gfCNCPoint4[12082] = {X 126.3568, Y 92.7333, Z -5.5000, A 0.000, B 0.000, C 0.000 }
gfCNCPoint4[12083] = {X 127.2181, Y 92.5238, Z -5.5000, A 0.000, B 0.000, C 0.000 }
gfCNCPoint4[12084] = {X 128.4710, Y 91.3461, Z -5.5000, A 0.000, B 0.000, C 0.000 }
gfCNCPoint4[12085] = {X 129.6569, Y 90.1009, Z -5.5000, A 0.000, B 0.000, C 0.000 }
gfCNCPoint4[12086] = {X 140.8575, Y 77.8010, Z -5.5000, A 0.000, B 0.000, C 0.000 }
gfCNCPoint4[12087] = {X 137.8975, Y 75.1055, Z -5.5000, A 0.000, B 0.000, C 0.000 }
gfCNCPoint4[12088] = {X 137.8979, Y 75.1051, Z -5.5000, A 0.000, B 0.000, C 0.000 }
gfCNCPoint4[12089] = {X 140.9141, Y 77.8526, Z -5.5000, A 0.000, B 0.000, C 0.000 }
gfCNCPoint4[12090] = {X 156.0371, Y 61.2507, Z -5.5000, A 0.000, B 0.000, C 0.000 }
gfCNCPoint4[12091] = {X 155.6323, Y 60.5351, Z -5.5000, A 0.000, B 0.000, C 0.000 }
gfCNCPoint4[12092] = {X 155.3824, Y 59.7518, Z -5.5000, A 0.000, B 0.000, C 0.000 }
gfCNCPoint4[12093] = {X 155.2980, Y 58.9341, Z -5.5000, A 0.000, B 0.000, C 0.000 }
gfCNCPoint4[12094] = {X 155.2980, Y 58.0000, Z -5.5000, A 0.000, B 0.000, C 0.000 }
gfCNCPoint4[12095] = {X 155.3982, Y 57.1099, Z -5.5000, A 0.000, B 0.000, C 0.000 }
gfCNCPoint4[12096] = {X 155.6941, Y 56.2645, Z -5.5000, A 0.000, B 0.000, C 0.000 }
gfCNCPoint4[12097] = {X 156.1706, Y 55.5060, Z -5.5000, A 0.000, B 0.000, C 0.000 }
gfCNCPoint4[12098] = {X 156.8040, Y 54.8727, Z -5.5000, A 0.000, B 0.000, C 0.000 }
gfCNCPoint4[12099] = {X 157.5624, Y 54.3961, Z -5.5000, A 0.000, B 0.000, C 0.000 }
gfCNCPoint4[12100] = {X 158.4079, Y 54.1003, Z -5.5000, A 0.000, B 0.000, C 0.000 }
gfCNCPoint4[12101] = {X 159.2980, Y 54.0000, Z -5.5000, A 0.000, B 0.000, C 0.000 }
gfCNCPoint4[12102] = {X 178.5335, Y 54.0000, Z -5.5000, A 0.000, B 0.000, C 0.000 }
gfCNCPoint4[12103] = {X 179.4236, Y 54.1003, Z -5.5000, A 0.000, B 0.000, C 0.000 }
gfCNCPoint4[12104] = {X 180.2690, Y 54.3961, Z -5.5000, A 0.000, B 0.000, C 0.000 }
gfCNCPoint4[12105] = {X 181.0275, Y 54.8727, Z -5.5000, A 0.000, B 0.000, C 0.000 }
gfCNCPoint4[12106] = {X 181.6608, Y 55.5060, Z -5.5000, A 0.000, B 0.000, C 0.000 }
gfCNCPoint4[12107] = {X 182.1374, Y 56.2645, Z -5.5000, A 0.000, B 0.000, C 0.000 }
gfCNCPoint4[12108] = {X 182.4332, Y 57.1099, Z -5.5000, A 0.000, B 0.000, C 0.000 }
gfCNCPoint4[12109] = {X 182.5335, Y 58.0000, Z -5.5000, A 0.000, B 0.000, C 0.000 }
gfCNCPoint4[12110] = {X 182.5334, Y 58.9671, Z -5.5000, A 0.000, B 0.000, C 0.000 }
gfCNCPoint4[12111] = {X 182.4463, Y 59.7646, Z -5.5000, A 0.000, B 0.000, C 0.000 }
gfCNCPoint4[12112] = {X 182.2019, Y 60.5286, Z -5.5000, A 0.000, B 0.000, C 0.000 }
gfCNCPoint4[12113] = {X 181.8100, Y 61.2285, Z -5.5000, A 0.000, B 0.000, C 0.000 }
gfCNCPoint4[12114] = {X 209.2433, Y 91.1704, Z -5.5000, A 0.000, B 0.000, C 0.000 }
gfCNCPoint4[12115] = {X 209.9164, Y 91.8534, Z -5.5000, A 0.000, B 0.000, C 0.000 }
gfCNCPoint4[12116] = {X 210.6375, Y 92.4856, Z -5.5000, A 0.000, B 0.000, C 0.000 }
gfCNCPoint4[12117] = {X 210.9790, Y 92.7012, Z -5.5000, A 0.000, B 0.000, C 0.000 }
gfCNCPoint4[12118] = {X 211.3621, Y 92.8295, Z -5.5000, A 0.000, B 0.000, C 0.000 }
gfCNCPoint4[12119] = {X 212.0545, Y 92.9775, Z -5.5000, A 0.000, B 0.000, C 0.000 }
gfCNCPoint4[12120] = {X 213.3961, Y 93.1465, Z -5.5000, A 0.000, B 0.000, C 0.000 }
gfCNCPoint4[12121] = {X 214.4555, Y 93.0562, Z -5.5000, A 0.000, B 0.000, C 0.000 }
gfCNCPoint4[12122] = {X 215.5170, Y 92.9951, Z -5.5000, A 0.000, B 0.000, C 0.000 }
gfCNCPoint4[12123] = {X 216.2444, Y 92.9150, Z -5.5000, A 0.000, B 0.000, C 0.000 }
gfCNCPoint4[12124] = {X 216.9448, Y 92.7028, Z -5.5000, A 0.000, B 0.000, C 0.000 }
gfCNCPoint4[12125] = {X 217.5944, Y 92.3657, Z -5.5000, A 0.000, B 0.000, C 0.000 }
gfCNCPoint4[12126] = {X 223.1343, Y 88.7905, Z -5.5000, A 0.000, B 0.000, C 0.000 }
gfCNCPoint4[12127] = {X 246.5290, Y 73.8310, Z -5.5000, A 0.000, B 0.000, C 0.000 }
gfCNCPoint4[12128] = {X 221.7493, Y 64.1069, Z -5.5000, A 0.000, B 0.000, C 0.000 }
gfCNCPoint4[12129] = {X 219.9471, Y 63.5037, Z -5.5000, A 0.000, B 0.000, C 0.000 }
gfCNCPoint4[12130] = {X 218.0879, Y 63.1103, Z -5.5000, A 0.000, B 0.000, C 0.000 }
gfCNCPoint4[12131] = {X 216.1958, Y 62.9318, Z -5.5000, A 0.000, B 0.000, C 0.000 }
gfCNCPoint4[12132] = {X 215.3283, Y 62.8064, Z -5.5000, A 0.000, B 0.000, C 0.000 }
gfCNCPoint4[12133] = {X 214.5089, Y 62.4951, Z -5.5000, A 0.000, B 0.000, C 0.000 }
gfCNCPoint4[12134] = {X 213.7770, Y 62.0127, Z -5.5000, A 0.000, B 0.000, C 0.000 }
gfCNCPoint4[12135] = {X 213.1677, Y 61.3825, Z -5.5000, A 0.000, B 0.000, C 0.000 }
gfCNCPoint4[12136] = {X 212.7104, Y 60.6348, Z -5.5000, A 0.000, B 0.000, C 0.000 }
gfCNCPoint4[12137] = {X 212.4268, Y 59.8053, Z -5.5000, A 0.000, B 0.000, C 0.000 }
gfCNCPoint4[12138] = {X 212.3308, Y 58.9341, Z -5.5000, A 0.000, B 0.000, C 0.000 }
gfCNCPoint4[12139] = {X 212.3308, Y 58.0000, Z -5.5000, A 0.000, B 0.000, C 0.000 }
gfCNCPoint4[12140] = {X 212.4311, Y 57.1099, Z -5.5000, A 0.000, B 0.000, C 0.000 }
gfCNCPoint4[12141] = {X 212.7269, Y 56.2645, Z -5.5000, A 0.000, B 0.000, C 0.000 }
gfCNCPoint4[12142] = {X 213.2035, Y 55.5060, Z -5.5000, A 0.000, B 0.000, C 0.000 }
gfCNCPoint4[12143] = {X 213.8368, Y 54.8727, Z -5.5000, A 0.000, B 0.000, C 0.000 }
gfCNCPoint4[12144] = {X 214.5953, Y 54.3961, Z -5.5000, A 0.000, B 0.000, C 0.000 }
gfCNCPoint4[12145] = {X 215.4407, Y 54.1003, Z -5.5000, A 0.000, B 0.000, C 0.000 }
gfCNCPoint4[12146] = {X 216.3308, Y 54.0000, Z -5.5000, A 0.000, B 0.000, C 0.000 }
gfCNCPoint4[12147] = {X 237.2617, Y 54.0000, Z -5.5000, A 0.000, B 0.000, C 0.000 }
gfCNCPoint4[12148] = {X 238.1518, Y 54.1003, Z -5.5000, A 0.000, B 0.000, C 0.000 }
gfCNCPoint4[12149] = {X 238.9972, Y 54.3961, Z -5.5000, A 0.000, B 0.000, C 0.000 }
gfCNCPoint4[12150] = {X 239.7556, Y 54.8727, Z -5.5000, A 0.000, B 0.000, C 0.000 }
gfCNCPoint4[12151] = {X 240.3890, Y 55.5060, Z -5.5000, A 0.000, B 0.000, C 0.000 }
gfCNCPoint4[12152] = {X 240.8656, Y 56.2645, Z -5.5000, A 0.000, B 0.000, C 0.000 }
gfCNCPoint4[12153] = {X 241.1614, Y 57.1099, Z -5.5000, A 0.000, B 0.000, C 0.000 }
gfCNCPoint4[12154] = {X 241.2617, Y 58.0000, Z -5.5000, A 0.000, B 0.000, C 0.000 }
gfCNCPoint4[12155] = {X 241.2617, Y 58.4508, Z -5.5000, A 0.000, B 0.000, C 0.000 }
gfCNCPoint4[12156] = {X 247.9970, Y 61.0771, Z -5.5000, A 0.000, B 0.000, C 0.000 }
gfCNCPoint4[12157] = {X 275.9525, Y 72.1731, Z -5.5000, A 0.000, B 0.000, C 0.000 }
gfCNCPoint4[12158] = {X 275.9520, Y 63.0389, Z -5.5000, A 0.000, B 0.000, C 0.000 }
gfCNCPoint4[12159] = {X 275.9573, Y 62.9246, Z -5.5000, A 0.000, B 0.000, C 0.000 }
gfCNCPoint4[12160] = {X 275.7852, Y 62.9090, Z -5.5000, A 0.000, B 0.000, C 0.000 }
gfCNCPoint4[12161] = {X 275.6139, Y 62.8859, Z -5.5000, A 0.000, B 0.000, C 0.000 }
gfCNCPoint4[12162] = {X 274.7074, Y 62.6318, Z -5.5000, A 0.000, B 0.000, C 0.000 }
gfCNCPoint4[12163] = {X 273.8854, Y 62.1729, Z -5.5000, A 0.000, B 0.000, C 0.000 }
gfCNCPoint4[12164] = {X 273.1934, Y 61.5345, Z -5.5000, A 0.000, B 0.000, C 0.000 }
gfCNCPoint4[12165] = {X 272.6697, Y 60.7521, Z -5.5000, A 0.000, B 0.000, C 0.000 }
gfCNCPoint4[12166] = {X 272.3435, Y 59.8690, Z -5.5000, A 0.000, B 0.000, C 0.000 }
gfCNCPoint4[12167] = {X 272.2327, Y 58.9341, Z -5.5000, A 0.000, B 0.000, C 0.000 }
gfCNCPoint4[12168] = {X 272.2327, Y 58.0000, Z -5.5000, A 0.000, B 0.000, C 0.000 }
gfCNCPoint4[12169] = {X 272.3330, Y 57.1099, Z -5.5000, A 0.000, B 0.000, C 0.000 }
gfCNCPoint4[12170] = {X 272.6288, Y 56.2645, Z -5.5000, A 0.000, B 0.000, C 0.000 }
gfCNCPoint4[12171] = {X 273.1054, Y 55.5060, Z -5.5000, A 0.000, B 0.000, C 0.000 }
gfCNCPoint4[12172] = {X 273.7387, Y 54.8727, Z -5.5000, A 0.000, B 0.000, C 0.000 }
gfCNCPoint4[12173] = {X 274.4972, Y 54.3961, Z -5.5000, A 0.000, B 0.000, C 0.000 }
gfCNCPoint4[12174] = {X 275.3426, Y 54.1003, Z -5.5000, A 0.000, B 0.000, C 0.000 }
gfCNCPoint4[12175] = {X 276.2327, Y 54.0000, Z -5.5000, A 0.000, B 0.000, C 0.000 }
gfCNCPoint4[12176] = {X 292.7731, Y 54.0000, Z -5.5000, A 0.000, B 0.000, C 0.000 }
gfCNCPoint4[12177] = {X 293.6632, Y 54.1003, Z -5.5000, A 0.000, B 0.000, C 0.000 }
gfCNCPoint4[12178] = {X 294.5086, Y 54.3961, Z -5.5000, A 0.000, B 0.000, C 0.000 }
gfCNCPoint4[12179] = {X 295.2670, Y 54.8727, Z -5.5000, A 0.000, B 0.000, C 0.000 }
gfCNCPoint4[12180] = {X 295.9004, Y 55.5060, Z -5.5000, A 0.000, B 0.000, C 0.000 }
gfCNCPoint4[12181] = {X 296.3770, Y 56.2645, Z -5.5000, A 0.000, B 0.000, C 0.000 }
gfCNCPoint4[12182] = {X 296.6728, Y 57.1099, Z -5.5000, A 0.000, B 0.000, C 0.000 }
gfCNCPoint4[12183] = {X 296.7731, Y 58.0000, Z -5.5000, A 0.000, B 0.000, C 0.000 }
gfCNCPoint4[12184] = {X 296.7731, Y 58.9341, Z -5.5000, A 0.000, B 0.000, C 0.000 }
gfCNCPoint4[12185] = {X 296.6600, Y 59.8686, Z -5.5000, A 0.000, B 0.000, C 0.000 }
gfCNCPoint4[12186] = {X 296.3325, Y 60.7511, Z -5.5000, A 0.000, B 0.000, C 0.000 }
gfCNCPoint4[12187] = {X 295.8085, Y 61.5331, Z -5.5000, A 0.000, B 0.000, C 0.000 }
gfCNCPoint4[12188] = {X 295.1170, Y 62.1717, Z -5.5000, A 0.000, B 0.000, C 0.000 }
gfCNCPoint4[12189] = {X 294.2958, Y 62.6318, Z -5.5000, A 0.000, B 0.000, C 0.000 }
gfCNCPoint4[12190] = {X 293.3900, Y 62.8882, Z -5.5000, A 0.000, B 0.000, C 0.000 }
gfCNCPoint4[12191] = {X 293.2330, Y 62.9101, Z -5.5000, A 0.000, B 0.000, C 0.000 }
gfCNCPoint4[12192] = {X 293.0752, Y 62.9258, Z -5.5000, A 0.000, B 0.000, C 0.000 }
gfCNCPoint4[12193] = {X 293.0531, Y 63.1540, Z -5.5000, A 0.000, B 0.000, C 0.000 }
gfCNCPoint4[12194] = {X 293.0531, Y 92.9237, Z -5.5000, A 0.000, B 0.000, C 0.000 }
gfCNCPoint4[12195] = {X 293.0752, Y 93.0668, Z -5.5000, A 0.000, B 0.000, C 0.000 }
gfCNCPoint4[12196] = {X 293.2324, Y 93.0830, Z -5.5000, A 0.000, B 0.000, C 0.000 }
gfCNCPoint4[12197] = {X 293.3888, Y 93.1053, Z -5.5000, A 0.000, B 0.000, C 0.000 }
gfCNCPoint4[12198] = {X 294.2943, Y 93.3643, Z -5.5000, A 0.000, B 0.000, C 0.000 }
gfCNCPoint4[12199] = {X 295.1151, Y 93.8262, Z -5.5000, A 0.000, B 0.000, C 0.000 }
gfCNCPoint4[12200] = {X 295.8064, Y 94.4658, Z -5.5000, A 0.000, B 0.000, C 0.000 }
gfCNCPoint4[12201] = {X 296.3304, Y 95.2484, Z -5.5000, A 0.000, B 0.000, C 0.000 }
gfCNCPoint4[12202] = {X 296.6586, Y 96.1312, Z -5.5000, A 0.000, B 0.000, C 0.000 }
gfCNCPoint4[12203] = {X 296.7731, Y 97.0661, Z -5.5000, A 0.000, B 0.000, C 0.000 }
gfCNCPoint4[12204] = {X 296.7731, Y 98.0000, Z -5.5000, A 0.000, B 0.000, C 0.000 }
gfCNCPoint4[12205] = {X 296.6728, Y 98.8901, Z -5.5000, A 0.000, B 0.000, C 0.000 }
gfCNCPoint4[12206] = {X 296.3770, Y 99.7355, Z -5.5000, A 0.000, B 0.000, C 0.000 }
gfCNCPoint4[12207] = {X 295.9004, Y 100.4940, Z -5.5000, A 0.000, B 0.000, C 0.000 }
gfCNCPoint4[12208] = {X 295.2670, Y 101.1273, Z -5.5000, A 0.000, B 0.000, C 0.000 }
gfCNCPoint4[12209] = {X 294.5086, Y 101.6039, Z -5.5000, A 0.000, B 0.000, C 0.000 }
gfCNCPoint4[12210] = {X 293.6632, Y 101.8997, Z -5.5000, A 0.000, B 0.000, C 0.000 }
gfCNCPoint4[12211] = {X 292.7731, Y 102.0000, Z -5.5000, A 0.000, B 0.000, C 0.000 }
gfCNCPoint4[12212] = {X 276.2327, Y 102.0000, Z -5.5000, A 0.000, B 0.000, C 0.000 }
gfCNCPoint4[12213] = {X 275.3426, Y 101.8997, Z -5.5000, A 0.000, B 0.000, C 0.000 }
gfCNCPoint4[12214] = {X 274.4972, Y 101.6039, Z -5.5000, A 0.000, B 0.000, C 0.000 }
gfCNCPoint4[12215] = {X 273.7387, Y 101.1273, Z -5.5000, A 0.000, B 0.000, C 0.000 }
gfCNCPoint4[12216] = {X 273.1054, Y 100.4940, Z -5.5000, A 0.000, B 0.000, C 0.000 }
gfCNCPoint4[12217] = {X 272.6288, Y 99.7355, Z -5.5000, A 0.000, B 0.000, C 0.000 }
gfCNCPoint4[12218] = {X 272.3330, Y 98.8901, Z -5.5000, A 0.000, B 0.000, C 0.000 }
gfCNCPoint4[12219] = {X 272.2327, Y 98.0000, Z -5.5000, A 0.000, B 0.000, C 0.000 }
gfCNCPoint4[12220] = {X 272.2329, Y 97.0232, Z -5.5000, A 0.000, B 0.000, C 0.000 }
gfCNCPoint4[12221] = {X 272.3321, Y 96.1797, Z -5.5000, A 0.000, B 0.000, C 0.000 }
gfCNCPoint4[12222] = {X 272.6072, Y 95.3761, Z -5.5000, A 0.000, B 0.000, C 0.000 }
gfCNCPoint4[12223] = {X 273.0457, Y 94.6486, Z -5.5000, A 0.000, B 0.000, C 0.000 }
gfCNCPoint4[12224] = {X 273.6280, Y 94.0302, Z -5.5000, A 0.000, B 0.000, C 0.000 }
gfCNCPoint4[12225] = {X 274.3277, Y 93.5487, Z -5.5000, A 0.000, B 0.000, C 0.000 }
gfCNCPoint4[12226] = {X 275.1133, Y 93.2258, Z -5.5000, A 0.000, B 0.000, C 0.000 }
gfCNCPoint4[12227] = {X 275.9494, Y 93.0760, Z -5.5000, A 0.000, B 0.000, C 0.000 }
gfCNCPoint4[12228] = {X 275.9494, Y 85.3767, Z -5.5000, A 0.000, B 0.000, C 0.000 }
gfCNCPoint4[12229] = {X 262.6059, Y 80.1460, Z -5.5000, A 0.000, B 0.000, C 0.000 }
gfCNCPoint4[12230] = {X 262.1050, Y 80.4620, Z -5.5000, A 0.000, B 0.000, C 0.000 }
gfCNCPoint4[12231] = {X 237.4759, Y 96.4149, Z -5.5000, A 0.000, B 0.000, C 0.000 }
gfCNCPoint4[12232] = {X 237.4798, Y 97.0659, Z -5.5000, A 0.000, B 0.000, C 0.000 }
gfCNCPoint4[12233] = {X 237.4798, Y 98.0000, Z -5.5000, A 0.000, B 0.000, C 0.000 }
gfCNCPoint4[12234] = {X 237.3795, Y 98.8901, Z -5.5000, A 0.000, B 0.000, C 0.000 }
gfCNCPoint4[12235] = {X 237.0837, Y 99.7355, Z -5.5000, A 0.000, B 0.000, C 0.000 }
gfCNCPoint4[12236] = {X 236.6071, Y 100.4940, Z -5.5000, A 0.000, B 0.000, C 0.000 }
gfCNCPoint4[12237] = {X 235.9737, Y 101.1273, Z -5.5000, A 0.000, B 0.000, C 0.000 }
gfCNCPoint4[12238] = {X 235.2153, Y 101.6039, Z -5.5000, A 0.000, B 0.000, C 0.000 }
gfCNCPoint4[12239] = {X 234.3699, Y 101.8997, Z -5.5000, A 0.000, B 0.000, C 0.000 }
gfCNCPoint4[12240] = {X 233.4798, Y 102.0000, Z -5.5000, A 0.000, B 0.000, C 0.000 }
gfCNCPoint4[12241] = {X 214.1790, Y 102.0000, Z -5.5000, A 0.000, B 0.000, C 0.000 }
gfCNCPoint4[12242] = {X 213.7859, Y 101.9806, Z -5.5000, A 0.000, B 0.000, C 0.000 }
gfCNCPoint4[12243] = {X 213.3966, Y 101.9227, Z -5.5000, A 0.000, B 0.000, C 0.000 }
gfCNCPoint4[12244] = {X 213.0072, Y 101.9806, Z -5.5000, A 0.000, B 0.000, C 0.000 }
gfCNCPoint4[12245] = {X 212.6141, Y 102.0000, Z -5.5000, A 0.000, B 0.000, C 0.000 }
gfCNCPoint4[12246] = {X 194.9870, Y 102.0000, Z -5.5000, A 0.000, B 0.000, C 0.000 }
gfCNCPoint4[12247] = {X 194.0969, Y 101.8997, Z -5.5000, A 0.000, B 0.000, C 0.000 }
gfCNCPoint4[12248] = {X 193.2514, Y 101.6039, Z -5.5000, A 0.000, B 0.000, C 0.000 }
gfCNCPoint4[12249] = {X 192.4930, Y 101.1273, Z -5.5000, A 0.000, B 0.000, C 0.000 }
gfCNCPoint4[12250] = {X 191.8596, Y 100.4940, Z -5.5000, A 0.000, B 0.000, C 0.000 }
gfCNCPoint4[12251] = {X 191.3831, Y 99.7355, Z -5.5000, A 0.000, B 0.000, C 0.000 }
gfCNCPoint4[12252] = {X 191.0872, Y 98.8901, Z -5.5000, A 0.000, B 0.000, C 0.000 }
gfCNCPoint4[12253] = {X 190.9870, Y 98.0000, Z -5.5000, A 0.000, B 0.000, C 0.000 }
gfCNCPoint4[12254] = {X 190.9870, Y 97.0659, Z -5.5000, A 0.000, B 0.000, C 0.000 }
gfCNCPoint4[12255] = {X 191.0804, Y 96.2066, Z -5.5000, A 0.000, B 0.000, C 0.000 }
gfCNCPoint4[12256] = {X 191.3562, Y 95.3874, Z -5.5000, A 0.000, B 0.000, C 0.000 }
gfCNCPoint4[12257] = {X 191.8015, Y 94.6466, Z -5.5000, A 0.000, B 0.000, C 0.000 }
gfCNCPoint4[12258] = {X 191.9054, Y 94.5175, Z -5.5000, A 0.000, B 0.000, C 0.000 }
gfCNCPoint4[12259] = {X 192.0146, Y 94.3929, Z -5.5000, A 0.000, B 0.000, C 0.000 }
gfCNCPoint4[12260] = {X 188.7055, Y 90.7802, Z -5.5000, A 0.000, B 0.000, C 0.000 }
gfCNCPoint4[12261] = {X 149.9476, Y 90.7802, Z -5.5000, A 0.000, B 0.000, C 0.000 }
gfCNCPoint4[12262] = {X 146.7190, Y 94.3571, Z -5.5000, A 0.000, B 0.000, C 0.000 }
gfCNCPoint4[12263] = {X 147.1689, Y 94.9484, Z -5.5000, A 0.000, B 0.000, C 0.000 }
gfCNCPoint4[12264] = {X 147.5024, Y 95.6124, Z -5.5000, A 0.000, B 0.000, C 0.000 }
gfCNCPoint4[12265] = {X 147.7081, Y 96.3264, Z -5.5000, A 0.000, B 0.000, C 0.000 }
gfCNCPoint4[12266] = {X 147.7791, Y 97.0661, Z -5.5000, A 0.000, B 0.000, C 0.000 }
gfCNCPoint4[12267] = {X 147.7791, Y 98.0000, Z -5.5000, A 0.000, B 0.000, C 0.000 }
gfCNCPoint4[12268] = {X 147.6788, Y 98.8901, Z -5.5000, A 0.000, B 0.000, C 0.000 }
gfCNCPoint4[12269] = {X 147.3830, Y 99.7355, Z -5.5000, A 0.000, B 0.000, C 0.000 }
gfCNCPoint4[12270] = {X 146.9064, Y 100.4940, Z -5.5000, A 0.000, B 0.000, C 0.000 }
gfCNCPoint4[12271] = {X 146.2731, Y 101.1273, Z -5.5000, A 0.000, B 0.000, C 0.000 }
gfCNCPoint4[12272] = {X 145.5146, Y 101.6039, Z -5.5000, A 0.000, B 0.000, C 0.000 }
gfCNCPoint4[12273] = {X 144.6692, Y 101.8997, Z -5.5000, A 0.000, B 0.000, C 0.000 }
gfCNCPoint4[12274] = {X 143.7791, Y 102.0000, Z -5.5000, A 0.000, B 0.000, C 0.000 }
gfCNCPoint4[12275] = {X 125.0000, Y 102.0000, Z -5.5000, A 0.000, B 0.000, C 0.000 }
gfCNCPoint4[12276] = {X 124.1099, Y 101.8997, Z -5.5000, A 0.000, B 0.000, C 0.000 }
gfCNCPoint4[12277] = {X 123.2645, Y 101.6039, Z -5.5000, A 0.000, B 0.000, C 0.000 }
gfCNCPoint4[12278] = {X 122.5060, Y 101.1273, Z -5.5000, A 0.000, B 0.000, C 0.000 }
gfCNCPoint4[12279] = {X 121.8727, Y 100.4940, Z -5.5000, A 0.000, B 0.000, C 0.000 }
gfCNCPoint4[12280] = {X 121.3961, Y 99.7355, Z -5.5000, A 0.000, B 0.000, C 0.000 }
gfCNCPoint4[12281] = {X 121.1003, Y 98.8901, Z -5.5000, A 0.000, B 0.000, C 0.000 }
gfCNCPoint4[12282] = {X 121.0000, Y 98.0000, Z -5.5000, A 0.000, B 0.000, C 0.000 }
gfCNCPoint4[12283] = {X 121.0000, Y 97.0659, Z -5.5000, A 0.000, B 0.000, C 0.000 }
gfCNCPoint4[12284] = {X 121.0981, Y 96.1853, Z -5.5000, A 0.000, B 0.000, C 0.000 }
gfCNCPoint4[12285] = {X 121.3877, Y 95.3479, Z -5.5000, A 0.000, B 0.000, C 0.000 }
gfCNCPoint4[12286] = {X 121.8546, Y 94.5948, Z -5.5000, A 0.000, B 0.000, C 0.000 }
gfCNCPoint4[12287] = {X 122.4758, Y 93.9629, Z -5.5000, A 0.000, B 0.000, C 0.000 }
gfCNCPoint4[12288] = {X 123.2209, Y 93.4834, Z -5.5000, A 0.000, B 0.000, C 0.000 }
gfCNCPoint4[12289] = {X 124.0533, Y 93.1796, Z -5.5000, A 0.000, B 0.000, C 0.000 }
gfCNCPoint4[12290] = {X 124.9321, Y 93.0665, Z -5.5000, A 0.000, B 0.000, C 0.000 }
gfCNCPoint4[12291] = {X 124.9748, Y 93.0377, Z -5.5000, A 0.000, B 0.000, C 0.000 }
gfCNCPoint4[12292] = {X 125.4940, Y 92.9606, Z -5.5000, A 0.000, B 0.000, C 0.000 }
gfCNCPoint4[12293] = {X 126.3823, Y 92.8097, Z -5.5000, A 0.000, B 0.000, C 0.000 }
gfCNCPoint4[12294] = {X 127.2575, Y 92.5958, Z -5.5000, A 0.000, B 0.000, C 0.000 }
gfCNCPoint4[12295] = {X 128.5209, Y 91.4093, Z -5.5000, A 0.000, B 0.000, C 0.000 }
gfCNCPoint4[12296] = {X 129.7163, Y 90.1544, Z -5.5000, A 0.000, B 0.000, C 0.000 }
gfCNCPoint4[12297] = {X 133.8038, Y 85.6582, Z -5.5000, A 0.000, B 0.000, C 0.000 }
gfCNCPoint4[12298] = {X 140.9141, Y 77.8526, Z -5.5000, A 0.000, B 0.000, C 0.000 }
gfCNCPoint4[12299] = {X 137.8979, Y 75.1051, Z -5.5000, A 0.000, B 0.000, C 0.000 }
gfCNCPoint4[12300] = {X 137.8979, Y 75.1051, Z -2.5000, A 0.000, B 0.000, C 0.000 }
gfCNCPoint4[12301] = {X 137.8979, Y 75.1051, Z 11.0000, A 0.000, B 0.000, C 0.000 }
gfCNCPoint4[12302] = {X 165.2867, Y 38.5771, Z 11.0000, A 0.000, B 0.000, C 0.000 }
gfCNCPoint4[12303] = {X 165.2867, Y 38.5771, Z -2.5000, A 0.000, B 0.000, C 0.000 }
gfCNCPoint4[12304] = {X 165.2867, Y 38.5771, Z -5.5000, A 0.000, B 0.000, C 0.000 }
gfCNCPoint4[12305] = {X 169.3160, Y 37.9356, Z -5.5000, A 0.000, B 0.000, C 0.000 }
gfCNCPoint4[12306] = {X 169.2605, Y 37.5870, Z -5.5000, A 0.000, B 0.000, C 0.000 }
gfCNCPoint4[12307] = {X 169.1022, Y 35.9824, Z -5.5000, A 0.000, B 0.000, C 0.000 }
gfCNCPoint4[12308] = {X 169.1191, Y 34.3702, Z -5.5000, A 0.000, B 0.000, C 0.000 }
gfCNCPoint4[12309] = {X 169.3112, Y 32.7693, Z -5.5000, A 0.000, B 0.000, C 0.000 }
gfCNCPoint4[12310] = {X 169.6761, Y 31.1989, Z -5.5000, A 0.000, B 0.000, C 0.000 }
gfCNCPoint4[12311] = {X 170.2095, Y 29.6773, Z -5.5000, A 0.000, B 0.000, C 0.000 }
gfCNCPoint4[12312] = {X 170.8482, Y 28.3703, Z -5.5000, A 0.000, B 0.000, C 0.000 }
gfCNCPoint4[12313] = {X 171.6560, Y 27.1604, Z -5.5000, A 0.000, B 0.000, C 0.000 }
gfCNCPoint4[12314] = {X 172.6183, Y 26.0694, Z -5.5000, A 0.000, B 0.000, C 0.000 }
gfCNCPoint4[12315] = {X 173.7177, Y 25.1168, Z -5.5000, A 0.000, B 0.000, C 0.000 }
gfCNCPoint4[12316] = {X 174.9347, Y 24.3198, Z -5.5000, A 0.000, B 0.000, C 0.000 }
gfCNCPoint4[12317] = {X 174.1522, Y 23.9322, Z -5.5000, A 0.000, B 0.000, C 0.000 }
gfCNCPoint4[12318] = {X 173.4636, Y 23.3951, Z -5.5000, A 0.000, B 0.000, C 0.000 }
gfCNCPoint4[12319] = {X 172.8971, Y 22.7304, Z -5.5000, A 0.000, B 0.000, C 0.000 }
gfCNCPoint4[12320] = {X 172.4758, Y 21.9655, Z -5.5000, A 0.000, B 0.000, C 0.000 }
gfCNCPoint4[12321] = {X 169.8405, Y 15.5121, Z -5.5000, A 0.000, B 0.000, C 0.000 }
gfCNCPoint4[12322] = {X 169.5912, Y 14.6607, Z -5.5000, A 0.000, B 0.000, C 0.000 }
gfCNCPoint4[12323] = {X 169.5212, Y 13.7764, Z -5.5000, A 0.000, B 0.000, C 0.000 }
gfCNCPoint4[12324] = {X 169.6332, Y 12.8964, Z -5.5000, A 0.000, B 0.000, C 0.000 }
gfCNCPoint4[12325] = {X 169.9226, Y 12.0578, Z -5.5000, A 0.000, B 0.000, C 0.000 }
gfCNCPoint4[12326] = {X 170.3773, Y 11.2960, Z -5.5000, A 0.000, B 0.000, C 0.000 }
gfCNCPoint4[12327] = {X 170.9779, Y 10.6432, Z -5.5000, A 0.000, B 0.000, C 0.000 }
gfCNCPoint4[12328] = {X 171.6992, Y 10.1268, Z -5.5000, A 0.000, B 0.000, C 0.000 }
gfCNCPoint4[12329] = {X 172.3295, Y 9.7674, Z -5.5000, A 0.000, B 0.000, C 0.000 }
gfCNCPoint4[12330] = {X 173.1921, Y 9.4017, Z -5.5000, A 0.000, B 0.000, C 0.000 }
gfCNCPoint4[12331] = {X 174.1132, Y 9.2306, Z -5.5000, A 0.000, B 0.000, C 0.000 }
gfCNCPoint4[12332] = {X 175.0496, Y 9.2621, Z -5.5000, A 0.000, B 0.000, C 0.000 }
gfCNCPoint4[12333] = {X 175.9572, Y 9.4947, Z -5.5000, A 0.000, B 0.000, C 0.000 }
gfCNCPoint4[12334] = {X 177.1446, Y 9.0372, Z -5.5000, A 0.000, B 0.000, C 0.000 }
gfCNCPoint4[12335] = {X 179.3197, Y 8.2368, Z -5.5000, A 0.000, B 0.000, C 0.000 }
gfCNCPoint4[12336] = {X 181.5636, Y 7.6562, Z -5.5000, A 0.000, B 0.000, C 0.000 }
gfCNCPoint4[12337] = {X 183.8540, Y 7.3010, Z -5.5000, A 0.000, B 0.000, C 0.000 }
gfCNCPoint4[12338] = {X 186.1683, Y 7.1749, Z -5.5000, A 0.000, B 0.000, C 0.000 }
gfCNCPoint4[12339] = {X 188.4837, Y 7.2789, Z -5.5000, A 0.000, B 0.000, C 0.000 }
gfCNCPoint4[12340] = {X 190.7774, Y 7.6122, Z -5.5000, A 0.000, B 0.000, C 0.000 }
gfCNCPoint4[12341] = {X 192.3552, Y 8.0008, Z -5.5000, A 0.000, B 0.000, C 0.000 }
gfCNCPoint4[12342] = {X 193.8890, Y 8.5372, Z -5.5000, A 0.000, B 0.000, C 0.000 }
gfCNCPoint4[12343] = {X 195.3650, Y 9.2167, Z -5.5000, A 0.000, B 0.000, C 0.000 }
gfCNCPoint4[12344] = {X 196.7700, Y 10.0332, Z -5.5000, A 0.000, B 0.000, C 0.000 }
gfCNCPoint4[12345] = {X 198.0911, Y 10.9792, Z -5.5000, A 0.000, B 0.000, C 0.000 }
gfCNCPoint4[12346] = {X 199.1510, Y 11.9221, Z -5.5000, A 0.000, B 0.000, C 0.000 }
gfCNCPoint4[12347] = {X 200.1020, Y 12.9746, Z -5.5000, A 0.000, B 0.000, C 0.000 }
gfCNCPoint4[12348] = {X 200.9329, Y 14.1244, Z -5.5000, A 0.000, B 0.000, C 0.000 }
gfCNCPoint4[12349] = {X 201.6338, Y 15.3577, Z -5.5000, A 0.000, B 0.000, C 0.000 }
gfCNCPoint4[12350] = {X 202.1964, Y 16.6600, Z -5.5000, A 0.000, B 0.000, C 0.000 }
gfCNCPoint4[12351] = {X 202.6706, Y 18.3163, Z -5.5000, A 0.000, B 0.000, C 0.000 }
gfCNCPoint4[12352] = {X 202.9520, Y 20.0160, Z -5.5000, A 0.000, B 0.000, C 0.000 }
gfCNCPoint4[12353] = {X 203.0370, Y 21.7368, Z -5.5000, A 0.000, B 0.000, C 0.000 }
gfCNCPoint4[12354] = {X 202.9245, Y 23.4560, Z -5.5000, A 0.000, B 0.000, C 0.000 }
gfCNCPoint4[12355] = {X 202.6158, Y 25.1509, Z -5.5000, A 0.000, B 0.000, C 0.000 }
gfCNCPoint4[12356] = {X 202.1739, Y 26.5971, Z -5.5000, A 0.000, B 0.000, C 0.000 }
gfCNCPoint4[12357] = {X 201.5492, Y 27.9741, Z -5.5000, A 0.000, B 0.000, C 0.000 }
gfCNCPoint4[12358] = {X 200.7519, Y 29.2591, Z -5.5000, A 0.000, B 0.000, C 0.000 }
gfCNCPoint4[12359] = {X 199.7956, Y 30.4304, Z -5.5000, A 0.000, B 0.000, C 0.000 }
gfCNCPoint4[12360] = {X 198.6960, Y 31.4685, Z -5.5000, A 0.000, B 0.000, C 0.000 }
gfCNCPoint4[12361] = {X 199.4973, Y 31.8097, Z -5.5000, A 0.000, B 0.000, C 0.000 }
gfCNCPoint4[12362] = {X 200.2138, Y 32.3047, Z -5.5000, A 0.000, B 0.000, C 0.000 }
gfCNCPoint4[12363] = {X 200.8164, Y 32.9334, Z -5.5000, A 0.000, B 0.000, C 0.000 }
gfCNCPoint4[12364] = {X 201.2808, Y 33.6702, Z -5.5000, A 0.000, B 0.000, C 0.000 }
gfCNCPoint4[12365] = {X 204.3222, Y 39.9530, Z -5.5000, A 0.000, B 0.000, C 0.000 }
gfCNCPoint4[12366] = {X 204.6427, Y 40.8622, Z -5.5000, A 0.000, B 0.000, C 0.000 }
gfCNCPoint4[12367] = {X 204.7537, Y 41.8197, Z -5.5000, A 0.000, B 0.000, C 0.000 }
gfCNCPoint4[12368] = {X 204.6496, Y 42.7781, Z -5.5000, A 0.000, B 0.000, C 0.000 }
gfCNCPoint4[12369] = {X 204.3355, Y 43.6895, Z -5.5000, A 0.000, B 0.000, C 0.000 }
gfCNCPoint4[12370] = {X 203.8272, Y 44.5085, Z -5.5000, A 0.000, B 0.000, C 0.000 }
gfCNCPoint4[12371] = {X 203.1499, Y 45.1945, Z -5.5000, A 0.000, B 0.000, C 0.000 }
gfCNCPoint4[12372] = {X 202.6137, Y 45.6280, Z -5.5000, A 0.000, B 0.000, C 0.000 }
gfCNCPoint4[12373] = {X 201.9093, Y 46.0919, Z -5.5000, A 0.000, B 0.000, C 0.000 }
gfCNCPoint4[12374] = {X 201.1282, Y 46.4105, Z -5.5000, A 0.000, B 0.000, C 0.000 }
gfCNCPoint4[12375] = {X 200.3002, Y 46.5717, Z -5.5000, A 0.000, B 0.000, C 0.000 }
gfCNCPoint4[12376] = {X 199.4567, Y 46.5693, Z -5.5000, A 0.000, B 0.000, C 0.000 }
gfCNCPoint4[12377] = {X 198.6296, Y 46.4035, Z -5.5000, A 0.000, B 0.000, C 0.000 }
gfCNCPoint4[12378] = {X 196.5191, Y 47.5044, Z -5.5000, A 0.000, B 0.000, C 0.000 }
gfCNCPoint4[12379] = {X 194.3239, Y 48.4248, Z -5.5000, A 0.000, B 0.000, C 0.000 }
gfCNCPoint4[12380] = {X 192.0593, Y 49.1582, Z -5.5000, A 0.000, B 0.000, C 0.000 }
gfCNCPoint4[12381] = {X 189.8462, Y 49.6708, Z -5.5000, A 0.000, B 0.000, C 0.000 }
gfCNCPoint4[12382] = {X 187.5926, Y 49.9566, Z -5.5000, A 0.000, B 0.000, C 0.000 }
gfCNCPoint4[12383] = {X 185.3216, Y 50.0128, Z -5.5000, A 0.000, B 0.000, C 0.000 }
gfCNCPoint4[12384] = {X 183.0566, Y 49.8389, Z -5.5000, A 0.000, B 0.000, C 0.000 }
gfCNCPoint4[12385] = {X 180.8209, Y 49.4365, Z -5.5000, A 0.000, B 0.000, C 0.000 }
gfCNCPoint4[12386] = {X 178.9809, Y 48.9032, Z -5.5000, A 0.000, B 0.000, C 0.000 }
gfCNCPoint4[12387] = {X 177.2146, Y 48.1613, Z -5.5000, A 0.000, B 0.000, C 0.000 }
gfCNCPoint4[12388] = {X 175.5456, Y 47.2208, Z -5.5000, A 0.000, B 0.000, C 0.000 }
gfCNCPoint4[12389] = {X 173.9962, Y 46.0942, Z -5.5000, A 0.000, B 0.000, C 0.000 }
gfCNCPoint4[12390] = {X 172.8554, Y 45.0534, Z -5.5000, A 0.000, B 0.000, C 0.000 }
gfCNCPoint4[12391] = {X 171.8458, Y 43.8849, Z -5.5000, A 0.000, B 0.000, C 0.000 }
gfCNCPoint4[12392] = {X 170.9816, Y 42.6051, Z -5.5000, A 0.000, B 0.000, C 0.000 }
gfCNCPoint4[12393] = {X 170.2749, Y 41.2320, Z -5.5000, A 0.000, B 0.000, C 0.000 }
gfCNCPoint4[12394] = {X 169.7357, Y 39.7849, Z -5.5000, A 0.000, B 0.000, C 0.000 }
gfCNCPoint4[12395] = {X 169.3715, Y 38.2842, Z -5.5000, A 0.000, B 0.000, C 0.000 }
gfCNCPoint4[12396] = {X 169.3160, Y 37.9356, Z -5.5000, A 0.000, B 0.000, C 0.000 }
gfCNCPoint4[12397] = {X 165.3657, Y 38.5645, Z -5.5000, A 0.000, B 0.000, C 0.000 }
gfCNCPoint4[12398] = {X 169.3950, Y 37.9230, Z -5.5000, A 0.000, B 0.000, C 0.000 }
gfCNCPoint4[12399] = {X 169.3395, Y 37.5748, Z -5.5000, A 0.000, B 0.000, C 0.000 }
gfCNCPoint4[12400] = {X 169.1821, Y 35.9789, Z -5.5000, A 0.000, B 0.000, C 0.000 }
gfCNCPoint4[12401] = {X 169.1990, Y 34.3753, Z -5.5000, A 0.000, B 0.000, C 0.000 }
gfCNCPoint4[12402] = {X 169.3900, Y 32.7831, Z -5.5000, A 0.000, B 0.000, C 0.000 }
gfCNCPoint4[12403] = {X 169.7529, Y 31.2210, Z -5.5000, A 0.000, B 0.000, C 0.000 }
gfCNCPoint4[12404] = {X 170.2835, Y 29.7077, Z -5.5000, A 0.000, B 0.000, C 0.000 }
gfCNCPoint4[12405] = {X 170.9353, Y 28.3795, Z -5.5000, A 0.000, B 0.000, C 0.000 }
gfCNCPoint4[12406] = {X 171.7629, Y 27.1530, Z -5.5000, A 0.000, B 0.000, C 0.000 }
gfCNCPoint4[12407] = {X 172.7507, Y 26.0515, Z -5.5000, A 0.000, B 0.000, C 0.000 }
gfCNCPoint4[12408] = {X 173.8801, Y 25.0957, Z -5.5000, A 0.000, B 0.000, C 0.000 }
gfCNCPoint4[12409] = {X 175.1297, Y 24.3035, Z -5.5000, A 0.000, B 0.000, C 0.000 }
gfCNCPoint4[12410] = {X 174.3083, Y 23.9333, Z -5.5000, A 0.000, B 0.000, C 0.000 }
gfCNCPoint4[12411] = {X 173.5836, Y 23.3980, Z -5.5000, A 0.000, B 0.000, C 0.000 }
gfCNCPoint4[12412] = {X 172.9885, Y 22.7216, Z -5.5000, A 0.000, B 0.000, C 0.000 }
gfCNCPoint4[12413] = {X 172.5496, Y 21.9347, Z -5.5000, A 0.000, B 0.000, C 0.000 }
gfCNCPoint4[12414] = {X 169.9145, Y 15.4818, Z -5.5000, A 0.000, B 0.000, C 0.000 }
gfCNCPoint4[12415] = {X 169.6699, Y 14.6462, Z -5.5000, A 0.000, B 0.000, C 0.000 }
gfCNCPoint4[12416] = {X 169.6011, Y 13.7783, Z -5.5000, A 0.000, B 0.000, C 0.000 }
gfCNCPoint4[12417] = {X 169.7111, Y 12.9146, Z -5.5000, A 0.000, B 0.000, C 0.000 }
gfCNCPoint4[12418] = {X 169.9952, Y 12.0915, Z -5.5000, A 0.000, B 0.000, C 0.000 }
gfCNCPoint4[12419] = {X 170.4414, Y 11.3439, Z -5.5000, A 0.000, B 0.000, C 0.000 }
gfCNCPoint4[12420] = {X 171.0309, Y 10.7031, Z -5.5000, A 0.000, B 0.000, C 0.000 }
gfCNCPoint4[12421] = {X 171.7389, Y 10.1963, Z -5.5000, A 0.000, B 0.000, C 0.000 }
gfCNCPoint4[12422] = {X 172.3689, Y 9.8371, Z -5.5000, A 0.000, B 0.000, C 0.000 }
gfCNCPoint4[12423] = {X 173.2227, Y 9.4761, Z -5.5000, A 0.000, B 0.000, C 0.000 }
gfCNCPoint4[12424] = {X 174.1345, Y 9.3093, Z -5.5000, A 0.000, B 0.000, C 0.000 }
gfCNCPoint4[12425] = {X 175.0609, Y 9.3446, Z -5.5000, A 0.000, B 0.000, C 0.000 }
gfCNCPoint4[12426] = {X 175.9574, Y 9.5804, Z -5.5000, A 0.000, B 0.000, C 0.000 }
gfCNCPoint4[12427] = {X 177.1746, Y 9.1113, Z -5.5000, A 0.000, B 0.000, C 0.000 }
gfCNCPoint4[12428] = {X 179.3425, Y 8.3135, Z -5.5000, A 0.000, B 0.000, C 0.000 }
gfCNCPoint4[12429] = {X 181.5789, Y 7.7347, Z -5.5000, A 0.000, B 0.000, C 0.000 }
gfCNCPoint4[12430] = {X 183.8616, Y 7.3807, Z -5.5000, A 0.000, B 0.000, C 0.000 }
gfCNCPoint4[12431] = {X 186.1682, Y 7.2549, Z -5.5000, A 0.000, B 0.000, C 0.000 }
gfCNCPoint4[12432] = {X 188.4760, Y 7.3586, Z -5.5000, A 0.000, B 0.000, C 0.000 }
gfCNCPoint4[12433] = {X 190.7620, Y 7.6907, Z -5.5000, A 0.000, B 0.000, C 0.000 }
gfCNCPoint4[12434] = {X 192.3324, Y 8.0775, Z -5.5000, A 0.000, B 0.000, C 0.000 }
gfCNCPoint4[12435] = {X 193.8590, Y 8.6114, Z -5.5000, A 0.000, B 0.000, C 0.000 }
gfCNCPoint4[12436] = {X 195.3282, Y 9.2877, Z -5.5000, A 0.000, B 0.000, C 0.000 }
gfCNCPoint4[12437] = {X 196.7265, Y 10.1003, Z -5.5000, A 0.000, B 0.000, C 0.000 }
gfCNCPoint4[12438] = {X 198.0415, Y 11.0419, Z -5.5000, A 0.000, B 0.000, C 0.000 }
gfCNCPoint4[12439] = {X 199.0948, Y 11.9790, Z -5.5000, A 0.000, B 0.000, C 0.000 }
gfCNCPoint4[12440] = {X 200.0399, Y 13.0251, Z -5.5000, A 0.000, B 0.000, C 0.000 }
gfCNCPoint4[12441] = {X 200.8656, Y 14.1678, Z -5.5000, A 0.000, B 0.000, C 0.000 }
gfCNCPoint4[12442] = {X 201.5622, Y 15.3935, Z -5.5000, A 0.000, B 0.000, C 0.000 }
gfCNCPoint4[12443] = {X 202.1213, Y 16.6876, Z -5.5000, A 0.000, B 0.000, C 0.000 }
gfCNCPoint4[12444] = {X 202.5928, Y 18.3350, Z -5.5000, A 0.000, B 0.000, C 0.000 }
gfCNCPoint4[12445] = {X 202.8726, Y 20.0254, Z -5.5000, A 0.000, B 0.000, C 0.000 }
gfCNCPoint4[12446] = {X 202.9570, Y 21.7368, Z -5.5000, A 0.000, B 0.000, C 0.000 }
gfCNCPoint4[12447] = {X 202.8450, Y 23.4466, Z -5.5000, A 0.000, B 0.000, C 0.000 }
gfCNCPoint4[12448] = {X 202.5380, Y 25.1323, Z -5.5000, A 0.000, B 0.000, C 0.000 }
gfCNCPoint4[12449] = {X 202.0884, Y 26.5970, Z -5.5000, A 0.000, B 0.000, C 0.000 }
gfCNCPoint4[12450] = {X 201.4500, Y 27.9897, Z -5.5000, A 0.000, B 0.000, C 0.000 }
gfCNCPoint4[12451] = {X 200.6338, Y 29.2862, Z -5.5000, A 0.000, B 0.000, C 0.000 }
gfCNCPoint4[12452] = {X 199.6541, Y 30.4641, Z -5.5000, A 0.000, B 0.000, C 0.000 }
gfCNCPoint4[12453] = {X 198.5278, Y 31.5027, Z -5.5000, A 0.000, B 0.000, C 0.000 }
gfCNCPoint4[12454] = {X 199.3591, Y 31.8267, Z -5.5000, A 0.000, B 0.000, C 0.000 }
gfCNCPoint4[12455] = {X 200.1042, Y 32.3174, Z -5.5000, A 0.000, B 0.000, C 0.000 }
gfCNCPoint4[12456] = {X 200.7301, Y 32.9531, Z -5.5000, A 0.000, B 0.000, C 0.000 }
gfCNCPoint4[12457] = {X 201.2091, Y 33.7058, Z -5.5000, A 0.000, B 0.000, C 0.000 }
gfCNCPoint4[12458] = {X 204.2502, Y 39.9879, Z -5.5000, A 0.000, B 0.000, C 0.000 }
gfCNCPoint4[12459] = {X 204.5648, Y 40.8802, Z -5.5000, A 0.000, B 0.000, C 0.000 }
gfCNCPoint4[12460] = {X 204.6737, Y 41.8200, Z -5.5000, A 0.000, B 0.000, C 0.000 }
gfCNCPoint4[12461] = {X 204.5715, Y 42.7606, Z -5.5000, A 0.000, B 0.000, C 0.000 }
gfCNCPoint4[12462] = {X 204.2633, Y 43.6551, Z -5.5000, A 0.000, B 0.000, C 0.000 }
gfCNCPoint4[12463] = {X 203.7643, Y 44.4590, Z -5.5000, A 0.000, B 0.000, C 0.000 }
gfCNCPoint4[12464] = {X 203.0996, Y 45.1323, Z -5.5000, A 0.000, B 0.000, C 0.000 }
gfCNCPoint4[12465] = {X 202.5634, Y 45.5658, Z -5.5000, A 0.000, B 0.000, C 0.000 }
gfCNCPoint4[12466] = {X 201.8658, Y 46.0244, Z -5.5000, A 0.000, B 0.000, C 0.000 }
gfCNCPoint4[12467] = {X 201.0921, Y 46.3378, Z -5.5000, A 0.000, B 0.000, C 0.000 }
gfCNCPoint4[12468] = {X 200.2720, Y 46.4940, Z -5.5000, A 0.000, B 0.000, C 0.000 }
gfCNCPoint4[12469] = {X 199.4372, Y 46.4869, Z -5.5000, A 0.000, B 0.000, C 0.000 }
gfCNCPoint4[12470] = {X 198.6199, Y 46.3168, Z -5.5000, A 0.000, B 0.000, C 0.000 }
gfCNCPoint4[12471] = {X 196.5061, Y 47.4222, Z -5.5000, A 0.000, B 0.000, C 0.000 }
gfCNCPoint4[12472] = {X 194.3068, Y 48.3458, Z -5.5000, A 0.000, B 0.000, C 0.000 }
gfCNCPoint4[12473] = {X 192.0376, Y 49.0812, Z -5.5000, A 0.000, B 0.000, C 0.000 }
gfCNCPoint4[12474] = {X 189.8323, Y 49.5920, Z -5.5000, A 0.000, B 0.000, C 0.000 }
gfCNCPoint4[12475] = {X 187.5867, Y 49.8768, Z -5.5000, A 0.000, B 0.000, C 0.000 }
gfCNCPoint4[12476] = {X 185.3237, Y 49.9329, Z -5.5000, A 0.000, B 0.000, C 0.000 }
gfCNCPoint4[12477] = {X 183.0667, Y 49.7595, Z -5.5000, A 0.000, B 0.000, C 0.000 }
gfCNCPoint4[12478] = {X 180.8389, Y 49.3586, Z -5.5000, A 0.000, B 0.000, C 0.000 }
gfCNCPoint4[12479] = {X 179.0076, Y 48.8278, Z -5.5000, A 0.000, B 0.000, C 0.000 }
gfCNCPoint4[12480] = {X 177.2498, Y 48.0895, Z -5.5000, A 0.000, B 0.000, C 0.000 }
gfCNCPoint4[12481] = {X 175.5888, Y 47.1534, Z -5.5000, A 0.000, B 0.000, C 0.000 }
gfCNCPoint4[12482] = {X 174.0467, Y 46.0322, Z -5.5000, A 0.000, B 0.000, C 0.000 }
gfCNCPoint4[12483] = {X 172.9129, Y 44.9978, Z -5.5000, A 0.000, B 0.000, C 0.000 }
gfCNCPoint4[12484] = {X 171.9096, Y 43.8366, Z -5.5000, A 0.000, B 0.000, C 0.000 }
gfCNCPoint4[12485] = {X 171.0507, Y 42.5648, Z -5.5000, A 0.000, B 0.000, C 0.000 }
gfCNCPoint4[12486] = {X 170.3483, Y 41.2003, Z -5.5000, A 0.000, B 0.000, C 0.000 }
gfCNCPoint4[12487] = {X 169.8124, Y 39.7622, Z -5.5000, A 0.000, B 0.000, C 0.000 }
gfCNCPoint4[12488] = {X 169.4504, Y 38.2708, Z -5.5000, A 0.000, B 0.000, C 0.000 }
gfCNCPoint4[12489] = {X 169.3950, Y 37.9230, Z -5.5000, A 0.000, B 0.000, C 0.000 }
gfCNCPoint4[12490] = {X 165.4447, Y 38.5520, Z -5.5000, A 0.000, B 0.000, C 0.000 }
gfCNCPoint4[12491] = {X 169.4740, Y 37.9104, Z -5.5000, A 0.000, B 0.000, C 0.000 }
gfCNCPoint4[12492] = {X 169.4186, Y 37.5626, Z -5.5000, A 0.000, B 0.000, C 0.000 }
gfCNCPoint4[12493] = {X 169.2620, Y 35.9753, Z -5.5000, A 0.000, B 0.000, C 0.000 }
gfCNCPoint4[12494] = {X 169.2788, Y 34.3805, Z -5.5000, A 0.000, B 0.000, C 0.000 }
gfCNCPoint4[12495] = {X 169.4688, Y 32.7968, Z -5.5000, A 0.000, B 0.000, C 0.000 }
gfCNCPoint4[12496] = {X 169.8298, Y 31.2432, Z -5.5000, A 0.000, B 0.000, C 0.000 }
gfCNCPoint4[12497] = {X 170.3575, Y 29.7381, Z -5.5000, A 0.000, B 0.000, C 0.000 }
gfCNCPoint4[12498] = {X 171.0239, Y 28.3862, Z -5.5000, A 0.000, B 0.000, C 0.000 }
gfCNCPoint4[12499] = {X 171.8738, Y 27.1414, Z -5.5000, A 0.000, B 0.000, C 0.000 }
gfCNCPoint4[12500] = {X 172.8902, Y 26.0284, Z -5.5000, A 0.000, B 0.000, C 0.000 }
gfCNCPoint4[12501] = {X 174.0529, Y 25.0694, Z -5.5000, A 0.000, B 0.000, C 0.000 }
gfCNCPoint4[12502] = {X 175.3388, Y 24.2832, Z -5.5000, A 0.000, B 0.000, C 0.000 }
gfCNCPoint4[12503] = {X 174.4746, Y 23.9352, Z -5.5000, A 0.000, B 0.000, C 0.000 }
gfCNCPoint4[12504] = {X 173.7096, Y 23.4035, Z -5.5000, A 0.000, B 0.000, C 0.000 }
gfCNCPoint4[12505] = {X 173.0820, Y 22.7149, Z -5.5000, A 0.000, B 0.000, C 0.000 }
gfCNCPoint4[12506] = {X 172.6235, Y 21.9039, Z -5.5000, A 0.000, B 0.000, C 0.000 }
gfCNCPoint4[12507] = {X 169.9886, Y 15.4516, Z -5.5000, A 0.000, B 0.000, C 0.000 }
gfCNCPoint4[12508] = {X 169.7252, Y 14.4911, Z -5.5000, A 0.000, B 0.000, C 0.000 }
gfCNCPoint4[12509] = {X 169.6977, Y 13.4954, Z -5.5000, A 0.000, B 0.000, C 0.000 }
gfCNCPoint4[12510] = {X 169.9076, Y 12.5218, Z -5.5000, A 0.000, B 0.000, C 0.000 }
gfCNCPoint4[12511] = {X 170.3429, Y 11.6260, Z -5.5000, A 0.000, B 0.000, C 0.000 }
gfCNCPoint4[12512] = {X 170.9787, Y 10.8594, Z -5.5000, A 0.000, B 0.000, C 0.000 }
gfCNCPoint4[12513] = {X 171.7785, Y 10.2658, Z -5.5000, A 0.000, B 0.000, C 0.000 }
gfCNCPoint4[12514] = {X 172.4082, Y 9.9068, Z -5.5000, A 0.000, B 0.000, C 0.000 }
gfCNCPoint4[12515] = {X 173.2458, Y 9.5527, Z -5.5000, A 0.000, B 0.000, C 0.000 }
gfCNCPoint4[12516] = {X 174.1404, Y 9.3891, Z -5.5000, A 0.000, B 0.000, C 0.000 }
gfCNCPoint4[12517] = {X 175.0492, Y 9.4237, Z -5.5000, A 0.000, B 0.000, C 0.000 }
gfCNCPoint4[12518] = {X 175.9287, Y 9.6551, Z -5.5000, A 0.000, B 0.000, C 0.000 }
gfCNCPoint4[12519] = {X 176.0179, Y 9.6905, Z -5.5000, A 0.000, B 0.000, C 0.000 }
gfCNCPoint4[12520] = {X 177.2059, Y 9.1850, Z -5.5000, A 0.000, B 0.000, C 0.000 }
gfCNCPoint4[12521] = {X 179.3664, Y 8.3899, Z -5.5000, A 0.000, B 0.000, C 0.000 }
gfCNCPoint4[12522] = {X 181.5950, Y 7.8131, Z -5.5000, A 0.000, B 0.000, C 0.000 }
gfCNCPoint4[12523] = {X 183.8699, Y 7.4602, Z -5.5000, A 0.000, B 0.000, C 0.000 }
gfCNCPoint4[12524] = {X 186.1686, Y 7.3349, Z -5.5000, A 0.000, B 0.000, C 0.000 }
gfCNCPoint4[12525] = {X 188.4684, Y 7.4382, Z -5.5000, A 0.000, B 0.000, C 0.000 }
gfCNCPoint4[12526] = {X 190.7466, Y 7.7692, Z -5.5000, A 0.000, B 0.000, C 0.000 }
gfCNCPoint4[12527] = {X 192.6941, Y 8.2734, Z -5.5000, A 0.000, B 0.000, C 0.000 }
gfCNCPoint4[12528] = {X 194.5682, Y 9.0048, Z -5.5000, A 0.000, B 0.000, C 0.000 }
gfCNCPoint4[12529] = {X 196.3424, Y 9.9530, Z -5.5000, A 0.000, B 0.000, C 0.000 }
gfCNCPoint4[12530] = {X 197.9919, Y 11.1047, Z -5.5000, A 0.000, B 0.000, C 0.000 }
gfCNCPoint4[12531] = {X 199.2838, Y 12.2860, Z -5.5000, A 0.000, B 0.000, C 0.000 }
gfCNCPoint4[12532] = {X 200.4034, Y 13.6319, Z -5.5000, A 0.000, B 0.000, C 0.000 }
gfCNCPoint4[12533] = {X 201.3298, Y 15.1173, Z -5.5000, A 0.000, B 0.000, C 0.000 }
gfCNCPoint4[12534] = {X 202.0460, Y 16.7147, Z -5.5000, A 0.000, B 0.000, C 0.000 }
gfCNCPoint4[12535] = {X 202.5149, Y 18.3531, Z -5.5000, A 0.000, B 0.000, C 0.000 }
gfCNCPoint4[12536] = {X 202.7931, Y 20.0344, Z -5.5000, A 0.000, B 0.000, C 0.000 }
gfCNCPoint4[12537] = {X 202.8770, Y 21.7366, Z -5.5000, A 0.000, B 0.000, C 0.000 }
gfCNCPoint4[12538] = {X 202.7656, Y 23.4371, Z -5.5000, A 0.000, B 0.000, C 0.000 }
gfCNCPoint4[12539] = {X 202.4602, Y 25.1137, Z -5.5000, A 0.000, B 0.000, C 0.000 }
gfCNCPoint4[12540] = {X 202.0022, Y 26.5984, Z -5.5000, A 0.000, B 0.000, C 0.000 }
gfCNCPoint4[12541] = {X 201.3489, Y 28.0081, Z -5.5000, A 0.000, B 0.000, C 0.000 }
gfCNCPoint4[12542] = {X 200.5120, Y 29.3172, Z -5.5000, A 0.000, B 0.000, C 0.000 }
gfCNCPoint4[12543] = {X 199.5068, Y 30.5019, Z -5.5000, A 0.000, B 0.000, C 0.000 }
gfCNCPoint4[12544] = {X 198.3515, Y 31.5408, Z -5.5000, A 0.000, B 0.000, C 0.000 }
gfCNCPoint4[12545] = {X 199.2149, Y 31.8441, Z -5.5000, A 0.000, B 0.000, C 0.000 }
gfCNCPoint4[12546] = {X 199.9910, Y 32.3289, Z -5.5000, A 0.000, B 0.000, C 0.000 }
gfCNCPoint4[12547] = {X 200.6424, Y 32.9717, Z -5.5000, A 0.000, B 0.000, C 0.000 }
gfCNCPoint4[12548] = {X 201.1375, Y 33.7414, Z -5.5000, A 0.000, B 0.000, C 0.000 }
gfCNCPoint4[12549] = {X 204.1781, Y 40.0227, Z -5.5000, A 0.000, B 0.000, C 0.000 }
gfCNCPoint4[12550] = {X 204.4868, Y 40.8982, Z -5.5000, A 0.000, B 0.000, C 0.000 }
gfCNCPoint4[12551] = {X 204.5937, Y 41.8203, Z -5.5000, A 0.000, B 0.000, C 0.000 }
gfCNCPoint4[12552] = {X 204.4934, Y 42.7431, Z -5.5000, A 0.000, B 0.000, C 0.000 }
gfCNCPoint4[12553] = {X 204.1910, Y 43.6208, Z -5.5000, A 0.000, B 0.000, C 0.000 }
gfCNCPoint4[12554] = {X 203.7015, Y 44.4095, Z -5.5000, A 0.000, B 0.000, C 0.000 }
gfCNCPoint4[12555] = {X 203.0493, Y 45.0700, Z -5.5000, A 0.000, B 0.000, C 0.000 }
gfCNCPoint4[12556] = {X 202.5131, Y 45.5035, Z -5.5000, A 0.000, B 0.000, C 0.000 }
gfCNCPoint4[12557] = {X 201.8225, Y 45.9568, Z -5.5000, A 0.000, B 0.000, C 0.000 }
gfCNCPoint4[12558] = {X 201.0560, Y 46.2650, Z -5.5000, A 0.000, B 0.000, C 0.000 }
gfCNCPoint4[12559] = {X 200.2439, Y 46.4161, Z -5.5000, A 0.000, B 0.000, C 0.000 }
gfCNCPoint4[12560] = {X 199.4179, Y 46.4043, Z -5.5000, A 0.000, B 0.000, C 0.000 }
gfCNCPoint4[12561] = {X 198.6104, Y 46.2298, Z -5.5000, A 0.000, B 0.000, C 0.000 }
gfCNCPoint4[12562] = {X 196.4933, Y 47.3398, Z -5.5000, A 0.000, B 0.000, C 0.000 }
gfCNCPoint4[12563] = {X 194.2898, Y 48.2668, Z -5.5000, A 0.000, B 0.000, C 0.000 }
gfCNCPoint4[12564] = {X 192.0159, Y 49.0042, Z -5.5000, A 0.000, B 0.000, C 0.000 }
gfCNCPoint4[12565] = {X 189.8185, Y 49.5132, Z -5.5000, A 0.000, B 0.000, C 0.000 }
gfCNCPoint4[12566] = {X 187.5808, Y 49.7970, Z -5.5000, A 0.000, B 0.000, C 0.000 }
gfCNCPoint4[12567] = {X 185.3258, Y 49.8529, Z -5.5000, A 0.000, B 0.000, C 0.000 }
gfCNCPoint4[12568] = {X 183.0768, Y 49.6802, Z -5.5000, A 0.000, B 0.000, C 0.000 }
gfCNCPoint4[12569] = {X 180.8568, Y 49.2806, Z -5.5000, A 0.000, B 0.000, C 0.000 }
gfCNCPoint4[12570] = {X 179.0344, Y 48.7524, Z -5.5000, A 0.000, B 0.000, C 0.000 }
gfCNCPoint4[12571] = {X 177.2849, Y 48.0176, Z -5.5000, A 0.000, B 0.000, C 0.000 }
gfCNCPoint4[12572] = {X 175.6319, Y 47.0861, Z -5.5000, A 0.000, B 0.000, C 0.000 }
gfCNCPoint4[12573] = {X 174.0972, Y 45.9702, Z -5.5000, A 0.000, B 0.000, C 0.000 }
gfCNCPoint4[12574] = {X 172.9705, Y 44.9423, Z -5.5000, A 0.000, B 0.000, C 0.000 }
gfCNCPoint4[12575] = {X 171.9734, Y 43.7883, Z -5.5000, A 0.000, B 0.000, C 0.000 }
gfCNCPoint4[12576] = {X 171.1198, Y 42.5245, Z -5.5000, A 0.000, B 0.000, C 0.000 }
gfCNCPoint4[12577] = {X 170.4217, Y 41.1685, Z -5.5000, A 0.000, B 0.000, C 0.000 }
gfCNCPoint4[12578] = {X 169.8891, Y 39.7395, Z -5.5000, A 0.000, B 0.000, C 0.000 }
gfCNCPoint4[12579] = {X 169.5292, Y 38.2574, Z -5.5000, A 0.000, B 0.000, C 0.000 }
gfCNCPoint4[12580] = {X 169.4740, Y 37.9104, Z -5.5000, A 0.000, B 0.000, C 0.000 }
gfCNCPoint4[12581] = {X 165.5237, Y 38.5394, Z -5.5000, A 0.000, B 0.000, C 0.000 }
gfCNCPoint4[12582] = {X 169.5530, Y 37.8979, Z -5.5000, A 0.000, B 0.000, C 0.000 }
gfCNCPoint4[12583] = {X 169.4977, Y 37.5505, Z -5.5000, A 0.000, B 0.000, C 0.000 }
gfCNCPoint4[12584] = {X 169.3419, Y 35.9718, Z -5.5000, A 0.000, B 0.000, C 0.000 }
gfCNCPoint4[12585] = {X 169.3586, Y 34.3856, Z -5.5000, A 0.000, B 0.000, C 0.000 }
gfCNCPoint4[12586] = {X 169.5476, Y 32.8106, Z -5.5000, A 0.000, B 0.000, C 0.000 }
gfCNCPoint4[12587] = {X 169.9067, Y 31.2654, Z -5.5000, A 0.000, B 0.000, C 0.000 }
gfCNCPoint4[12588] = {X 170.4315, Y 29.7684, Z -5.5000, A 0.000, B 0.000, C 0.000 }
gfCNCPoint4[12589] = {X 171.1146, Y 28.3897, Z -5.5000, A 0.000, B 0.000, C 0.000 }
gfCNCPoint4[12590] = {X 171.9899, Y 27.1242, Z -5.5000, A 0.000, B 0.000, C 0.000 }
gfCNCPoint4[12591] = {X 173.0388, Y 25.9985, Z -5.5000, A 0.000, B 0.000, C 0.000 }
gfCNCPoint4[12592] = {X 174.2395, Y 25.0363, Z -5.5000, A 0.000, B 0.000, C 0.000 }
gfCNCPoint4[12593] = {X 175.5667, Y 24.2577, Z -5.5000, A 0.000, B 0.000, C 0.000 }
gfCNCPoint4[12594] = {X 174.6547, Y 23.9379, Z -5.5000, A 0.000, B 0.000, C 0.000 }
gfCNCPoint4[12595] = {X 173.8435, Y 23.4126, Z -5.5000, A 0.000, B 0.000, C 0.000 }
gfCNCPoint4[12596] = {X 173.1786, Y 22.7112, Z -5.5000, A 0.000, B 0.000, C 0.000 }
gfCNCPoint4[12597] = {X 172.6973, Y 21.8731, Z -5.5000, A 0.000, B 0.000, C 0.000 }
gfCNCPoint4[12598] = {X 170.0626, Y 15.4213, Z -5.5000, A 0.000, B 0.000, C 0.000 }
gfCNCPoint4[12599] = {X 169.8043, Y 14.4793, Z -5.5000, A 0.000, B 0.000, C 0.000 }
gfCNCPoint4[12600] = {X 169.7773, Y 13.5028, Z -5.5000, A 0.000, B 0.000, C 0.000 }
gfCNCPoint4[12601] = {X 169.9832, Y 12.5479, Z -5.5000, A 0.000, B 0.000, C 0.000 }
gfCNCPoint4[12602] = {X 170.4102, Y 11.6694, Z -5.5000, A 0.000, B 0.000, C 0.000 }
gfCNCPoint4[12603] = {X 171.0337, Y 10.9174, Z -5.5000, A 0.000, B 0.000, C 0.000 }
gfCNCPoint4[12604] = {X 171.8181, Y 10.3353, Z -5.5000, A 0.000, B 0.000, C 0.000 }
gfCNCPoint4[12605] = {X 172.4475, Y 9.9764, Z -5.5000, A 0.000, B 0.000, C 0.000 }
gfCNCPoint4[12606] = {X 173.2690, Y 9.6292, Z -5.5000, A 0.000, B 0.000, C 0.000 }
gfCNCPoint4[12607] = {X 174.1463, Y 9.4688, Z -5.5000, A 0.000, B 0.000, C 0.000 }
gfCNCPoint4[12608] = {X 175.0375, Y 9.5029, Z -5.5000, A 0.000, B 0.000, C 0.000 }
gfCNCPoint4[12609] = {X 175.9000, Y 9.7298, Z -5.5000, A 0.000, B 0.000, C 0.000 }
gfCNCPoint4[12610] = {X 175.9653, Y 9.7555, Z -5.5000, A 0.000, B 0.000, C 0.000 }
gfCNCPoint4[12611] = {X 176.0301, Y 9.7823, Z -5.5000, A 0.000, B 0.000, C 0.000 }
gfCNCPoint4[12612] = {X 176.0579, Y 9.7604, Z -5.5000, A 0.000, B 0.000, C 0.000 }
gfCNCPoint4[12613] = {X 177.2373, Y 9.2586, Z -5.5000, A 0.000, B 0.000, C 0.000 }
gfCNCPoint4[12614] = {X 179.3902, Y 8.4662, Z -5.5000, A 0.000, B 0.000, C 0.000 }
gfCNCPoint4[12615] = {X 181.6112, Y 7.8914, Z -5.5000, A 0.000, B 0.000, C 0.000 }
gfCNCPoint4[12616] = {X 183.8783, Y 7.5398, Z -5.5000, A 0.000, B 0.000, C 0.000 }
gfCNCPoint4[12617] = {X 186.1690, Y 7.4149, Z -5.5000, A 0.000, B 0.000, C 0.000 }
gfCNCPoint4[12618] = {X 188.4608, Y 7.5178, Z -5.5000, A 0.000, B 0.000, C 0.000 }
gfCNCPoint4[12619] = {X 190.7311, Y 7.8477, Z -5.5000, A 0.000, B 0.000, C 0.000 }
gfCNCPoint4[12620] = {X 192.6695, Y 8.3496, Z -5.5000, A 0.000, B 0.000, C 0.000 }
gfCNCPoint4[12621] = {X 194.5347, Y 9.0775, Z -5.5000, A 0.000, B 0.000, C 0.000 }
gfCNCPoint4[12622] = {X 196.3006, Y 10.0212, Z -5.5000, A 0.000, B 0.000, C 0.000 }
gfCNCPoint4[12623] = {X 197.9423, Y 11.1674, Z -5.5000, A 0.000, B 0.000, C 0.000 }
gfCNCPoint4[12624] = {X 199.2260, Y 12.3413, Z -5.5000, A 0.000, B 0.000, C 0.000 }
gfCNCPoint4[12625] = {X 200.3384, Y 13.6786, Z -5.5000, A 0.000, B 0.000, C 0.000 }
gfCNCPoint4[12626] = {X 201.2590, Y 15.1545, Z -5.5000, A 0.000, B 0.000, C 0.000 }
gfCNCPoint4[12627] = {X 201.9707, Y 16.7417, Z -5.5000, A 0.000, B 0.000, C 0.000 }
gfCNCPoint4[12628] = {X 202.4370, Y 18.3713, Z -5.5000, A 0.000, B 0.000, C 0.000 }
gfCNCPoint4[12629] = {X 202.7136, Y 20.0435, Z -5.5000, A 0.000, B 0.000, C 0.000 }
gfCNCPoint4[12630] = {X 202.7970, Y 21.7363, Z -5.5000, A 0.000, B 0.000, C 0.000 }
gfCNCPoint4[12631] = {X 202.6861, Y 23.4276, Z -5.5000, A 0.000, B 0.000, C 0.000 }
gfCNCPoint4[12632] = {X 202.3824, Y 25.0951, Z -5.5000, A 0.000, B 0.000, C 0.000 }
gfCNCPoint4[12633] = {X 201.9152, Y 26.6018, Z -5.5000, A 0.000, B 0.000, C 0.000 }
gfCNCPoint4[12634] = {X 201.2454, Y 28.0300, Z -5.5000, A 0.000, B 0.000, C 0.000 }
gfCNCPoint4[12635] = {X 200.3857, Y 29.3527, Z -5.5000, A 0.000, B 0.000, C 0.000 }
gfCNCPoint4[12636] = {X 199.3525, Y 30.5447, Z -5.5000, A 0.000, B 0.000, C 0.000 }
gfCNCPoint4[12637] = {X 198.1653, Y 31.5835, Z -5.5000, A 0.000, B 0.000, C 0.000 }
gfCNCPoint4[12638] = {X 199.0631, Y 31.8622, Z -5.5000, A 0.000, B 0.000, C 0.000 }
gfCNCPoint4[12639] = {X 199.8733, Y 32.3391, Z -5.5000, A 0.000, B 0.000, C 0.000 }
gfCNCPoint4[12640] = {X 200.5529, Y 32.9887, Z -5.5000, A 0.000, B 0.000, C 0.000 }
gfCNCPoint4[12641] = {X 201.0657, Y 33.7766, Z -5.5000, A 0.000, B 0.000, C 0.000 }
gfCNCPoint4[12642] = {X 204.1061, Y 40.0576, Z -5.5000, A 0.000, B 0.000, C 0.000 }
gfCNCPoint4[12643] = {X 204.4089, Y 40.9162, Z -5.5000, A 0.000, B 0.000, C 0.000 }
gfCNCPoint4[12644] = {X 204.5137, Y 41.8206, Z -5.5000, A 0.000, B 0.000, C 0.000 }
gfCNCPoint4[12645] = {X 204.4154, Y 42.7257, Z -5.5000, A 0.000, B 0.000, C 0.000 }
gfCNCPoint4[12646] = {X 204.1188, Y 43.5864, Z -5.5000, A 0.000, B 0.000, C 0.000 }
gfCNCPoint4[12647] = {X 203.6387, Y 44.3600, Z -5.5000, A 0.000, B 0.000, C 0.000 }
gfCNCPoint4[12648] = {X 202.9990, Y 45.0078, Z -5.5000, A 0.000, B 0.000, C 0.000 }
gfCNCPoint4[12649] = {X 202.4628, Y 45.4413, Z -5.5000, A 0.000, B 0.000, C 0.000 }
gfCNCPoint4[12650] = {X 201.7791, Y 45.8891, Z -5.5000, A 0.000, B 0.000, C 0.000 }
gfCNCPoint4[12651] = {X 201.0201, Y 46.1921, Z -5.5000, A 0.000, B 0.000, C 0.000 }
gfCNCPoint4[12652] = {X 200.2159, Y 46.3382, Z -5.5000, A 0.000, B 0.000, C 0.000 }
gfCNCPoint4[12653] = {X 199.3988, Y 46.3215, Z -5.5000, A 0.000, B 0.000, C 0.000 }
gfCNCPoint4[12654] = {X 198.6012, Y 46.1427, Z -5.5000, A 0.000, B 0.000, C 0.000 }
gfCNCPoint4[12655] = {X 196.4806, Y 47.2573, Z -5.5000, A 0.000, B 0.000, C 0.000 }
gfCNCPoint4[12656] = {X 194.2729, Y 48.1877, Z -5.5000, A 0.000, B 0.000, C 0.000 }
gfCNCPoint4[12657] = {X 191.9942, Y 48.9272, Z -5.5000, A 0.000, B 0.000, C 0.000 }
gfCNCPoint4[12658] = {X 189.8046, Y 49.4344, Z -5.5000, A 0.000, B 0.000, C 0.000 }
gfCNCPoint4[12659] = {X 187.5748, Y 49.7173, Z -5.5000, A 0.000, B 0.000, C 0.000 }
gfCNCPoint4[12660] = {X 185.3279, Y 49.7729, Z -5.5000, A 0.000, B 0.000, C 0.000 }
gfCNCPoint4[12661] = {X 183.0869, Y 49.6008, Z -5.5000, A 0.000, B 0.000, C 0.000 }
gfCNCPoint4[12662] = {X 180.8748, Y 49.2027, Z -5.5000, A 0.000, B 0.000, C 0.000 }
gfCNCPoint4[12663] = {X 179.0611, Y 48.6770, Z -5.5000, A 0.000, B 0.000, C 0.000 }
gfCNCPoint4[12664] = {X 177.3201, Y 47.9457, Z -5.5000, A 0.000, B 0.000, C 0.000 }
gfCNCPoint4[12665] = {X 175.6750, Y 47.0187, Z -5.5000, A 0.000, B 0.000, C 0.000 }
gfCNCPoint4[12666] = {X 174.1477, Y 45.9081, Z -5.5000, A 0.000, B 0.000, C 0.000 }
gfCNCPoint4[12667] = {X 173.0281, Y 44.8867, Z -5.5000, A 0.000, B 0.000, C 0.000 }
gfCNCPoint4[12668] = {X 172.0372, Y 43.7401, Z -5.5000, A 0.000, B 0.000, C 0.000 }
gfCNCPoint4[12669] = {X 171.1889, Y 42.4842, Z -5.5000, A 0.000, B 0.000, C 0.000 }
gfCNCPoint4[12670] = {X 170.4952, Y 41.1368, Z -5.5000, A 0.000, B 0.000, C 0.000 }
gfCNCPoint4[12671] = {X 169.9658, Y 39.7167, Z -5.5000, A 0.000, B 0.000, C 0.000 }
gfCNCPoint4[12672] = {X 169.6081, Y 38.2440, Z -5.5000, A 0.000, B 0.000, C 0.000 }
gfCNCPoint4[12673] = {X 169.5530, Y 37.8979, Z -5.5000, A 0.000, B 0.000, C 0.000 }
gfCNCPoint4[12674] = {X 165.6027, Y 38.5268, Z -5.5000, A 0.000, B 0.000, C 0.000 }
gfCNCPoint4[12675] = {X 169.6320, Y 37.8853, Z -5.5000, A 0.000, B 0.000, C 0.000 }
gfCNCPoint4[12676] = {X 169.5767, Y 37.5383, Z -5.5000, A 0.000, B 0.000, C 0.000 }
gfCNCPoint4[12677] = {X 169.4218, Y 35.9683, Z -5.5000, A 0.000, B 0.000, C 0.000 }
gfCNCPoint4[12678] = {X 169.4385, Y 34.3907, Z -5.5000, A 0.000, B 0.000, C 0.000 }
gfCNCPoint4[12679] = {X 169.6265, Y 32.8243, Z -5.5000, A 0.000, B 0.000, C 0.000 }
gfCNCPoint4[12680] = {X 169.9835, Y 31.2876, Z -5.5000, A 0.000, B 0.000, C 0.000 }
gfCNCPoint4[12681] = {X 170.5055, Y 29.7988, Z -5.5000, A 0.000, B 0.000, C 0.000 }
gfCNCPoint4[12682] = {X 171.2082, Y 28.3887, Z -5.5000, A 0.000, B 0.000, C 0.000 }
gfCNCPoint4[12683] = {X 172.1133, Y 27.0992, Z -5.5000, A 0.000, B 0.000, C 0.000 }
gfCNCPoint4[12684] = {X 173.2005, Y 25.9590, Z -5.5000, A 0.000, B 0.000, C 0.000 }
gfCNCPoint4[12685] = {X 174.4456, Y 24.9936, Z -5.5000, A 0.000, B 0.000, C 0.000 }
gfCNCPoint4[12686] = {X 175.8207, Y 24.2247, Z -5.5000, A 0.000, B 0.000, C 0.000 }
gfCNCPoint4[12687] = {X 175.0299, Y 24.0137, Z -5.5000, A 0.000, B 0.000, C 0.000 }
gfCNCPoint4[12688] = {X 174.2986, Y 23.6461, Z -5.5000, A 0.000, B 0.000, C 0.000 }
gfCNCPoint4[12689] = {X 173.6574, Y 23.1374, Z -5.5000, A 0.000, B 0.000, C 0.000 }
gfCNCPoint4[12690] = {X 173.1332, Y 22.5088, Z -5.5000, A 0.000, B 0.000, C 0.000 }
gfCNCPoint4[12691] = {X 172.7479, Y 21.7866, Z -5.5000, A 0.000, B 0.000, C 0.000 }
gfCNCPoint4[12692] = {X 170.1367, Y 15.3911, Z -5.5000, A 0.000, B 0.000, C 0.000 }
gfCNCPoint4[12693] = {X 169.8835, Y 14.4675, Z -5.5000, A 0.000, B 0.000, C 0.000 }
gfCNCPoint4[12694] = {X 169.8570, Y 13.5102, Z -5.5000, A 0.000, B 0.000, C 0.000 }
gfCNCPoint4[12695] = {X 170.0588, Y 12.5740, Z -5.5000, A 0.000, B 0.000, C 0.000 }
gfCNCPoint4[12696] = {X 170.4774, Y 11.7127, Z -5.5000, A 0.000, B 0.000, C 0.000 }
gfCNCPoint4[12697] = {X 171.0888, Y 10.9755, Z -5.5000, A 0.000, B 0.000, C 0.000 }
gfCNCPoint4[12698] = {X 171.8578, Y 10.4048, Z -5.5000, A 0.000, B 0.000, C 0.000 }
gfCNCPoint4[12699] = {X 172.4867, Y 10.0462, Z -5.5000, A 0.000, B 0.000, C 0.000 }
gfCNCPoint4[12700] = {X 173.2920, Y 9.7058, Z -5.5000, A 0.000, B 0.000, C 0.000 }
gfCNCPoint4[12701] = {X 174.1521, Y 9.5486, Z -5.5000, A 0.000, B 0.000, C 0.000 }
gfCNCPoint4[12702] = {X 175.0258, Y 9.5820, Z -5.5000, A 0.000, B 0.000, C 0.000 }
gfCNCPoint4[12703] = {X 175.8713, Y 9.8044, Z -5.5000, A 0.000, B 0.000, C 0.000 }
gfCNCPoint4[12704] = {X 175.9571, Y 9.8385, Z -5.5000, A 0.000, B 0.000, C 0.000 }
gfCNCPoint4[12705] = {X 176.0421, Y 9.8746, Z -5.5000, A 0.000, B 0.000, C 0.000 }
gfCNCPoint4[12706] = {X 176.0990, Y 9.8299, Z -5.5000, A 0.000, B 0.000, C 0.000 }
gfCNCPoint4[12707] = {X 177.2686, Y 9.3322, Z -5.5000, A 0.000, B 0.000, C 0.000 }
gfCNCPoint4[12708] = {X 179.4141, Y 8.5426, Z -5.5000, A 0.000, B 0.000, C 0.000 }
gfCNCPoint4[12709] = {X 181.6274, Y 7.9698, Z -5.5000, A 0.000, B 0.000, C 0.000 }
gfCNCPoint4[12710] = {X 183.8866, Y 7.6194, Z -5.5000, A 0.000, B 0.000, C 0.000 }
gfCNCPoint4[12711] = {X 186.1694, Y 7.4949, Z -5.5000, A 0.000, B 0.000, C 0.000 }
gfCNCPoint4[12712] = {X 188.4533, Y 7.5975, Z -5.5000, A 0.000, B 0.000, C 0.000 }
gfCNCPoint4[12713] = {X 190.7157, Y 7.9262, Z -5.5000, A 0.000, B 0.000, C 0.000 }
gfCNCPoint4[12714] = {X 192.6449, Y 8.4257, Z -5.5000, A 0.000, B 0.000, C 0.000 }
gfCNCPoint4[12715] = {X 194.5013, Y 9.1501, Z -5.5000, A 0.000, B 0.000, C 0.000 }
gfCNCPoint4[12716] = {X 196.2588, Y 10.0894, Z -5.5000, A 0.000, B 0.000, C 0.000 }
gfCNCPoint4[12717] = {X 197.8927, Y 11.2302, Z -5.5000, A 0.000, B 0.000, C 0.000 }
gfCNCPoint4[12718] = {X 199.1681, Y 12.3966, Z -5.5000, A 0.000, B 0.000, C 0.000 }
gfCNCPoint4[12719] = {X 200.2735, Y 13.7253, Z -5.5000, A 0.000, B 0.000, C 0.000 }
gfCNCPoint4[12720] = {X 201.1882, Y 15.1917, Z -5.5000, A 0.000, B 0.000, C 0.000 }
gfCNCPoint4[12721] = {X 201.8954, Y 16.7687, Z -5.5000, A 0.000, B 0.000, C 0.000 }
gfCNCPoint4[12722] = {X 202.3590, Y 18.3894, Z -5.5000, A 0.000, B 0.000, C 0.000 }
gfCNCPoint4[12723] = {X 202.6341, Y 20.0525, Z -5.5000, A 0.000, B 0.000, C 0.000 }
gfCNCPoint4[12724] = {X 202.7170, Y 21.7361, Z -5.5000, A 0.000, B 0.000, C 0.000 }
gfCNCPoint4[12725] = {X 202.6067, Y 23.4182, Z -5.5000, A 0.000, B 0.000, C 0.000 }
gfCNCPoint4[12726] = {X 202.3046, Y 25.0766, Z -5.5000, A 0.000, B 0.000, C 0.000 }
gfCNCPoint4[12727] = {X 201.8270, Y 26.6077, Z -5.5000, A 0.000, B 0.000, C 0.000 }
gfCNCPoint4[12728] = {X 201.1388, Y 28.0565, Z -5.5000, A 0.000, B 0.000, C 0.000 }
gfCNCPoint4[12729] = {X 200.2537, Y 29.3941, Z -5.5000, A 0.000, B 0.000, C 0.000 }
gfCNCPoint4[12730] = {X 199.1893, Y 30.5938, Z -5.5000, A 0.000, B 0.000, C 0.000 }
gfCNCPoint4[12731] = {X 197.9667, Y 31.6320, Z -5.5000, A 0.000, B 0.000, C 0.000 }
gfCNCPoint4[12732] = {X 198.7283, Y 31.8160, Z -5.5000, A 0.000, B 0.000, C 0.000 }
gfCNCPoint4[12733] = {X 199.4395, Y 32.1450, Z -5.5000, A 0.000, B 0.000, C 0.000 }
gfCNCPoint4[12734] = {X 200.0728, Y 32.6063, Z -5.5000, A 0.000, B 0.000, C 0.000 }
gfCNCPoint4[12735] = {X 200.6041, Y 33.1822, Z -5.5000, A 0.000, B 0.000, C 0.000 }
gfCNCPoint4[12736] = {X 201.0129, Y 33.8507, Z -5.5000, A 0.000, B 0.000, C 0.000 }
gfCNCPoint4[12737] = {X 204.0341, Y 40.0925, Z -5.5000, A 0.000, B 0.000, C 0.000 }
gfCNCPoint4[12738] = {X 204.3309, Y 40.9342, Z -5.5000, A 0.000, B 0.000, C 0.000 }
gfCNCPoint4[12739] = {X 204.4337, Y 41.8209, Z -5.5000, A 0.000, B 0.000, C 0.000 }
gfCNCPoint4[12740] = {X 204.3373, Y 42.7082, Z -5.5000, A 0.000, B 0.000, C 0.000 }
gfCNCPoint4[12741] = {X 204.0465, Y 43.5521, Z -5.5000, A 0.000, B 0.000, C 0.000 }
gfCNCPoint4[12742] = {X 203.5758, Y 44.3105, Z -5.5000, A 0.000, B 0.000, C 0.000 }
gfCNCPoint4[12743] = {X 202.9487, Y 44.9456, Z -5.5000, A 0.000, B 0.000, C 0.000 }
gfCNCPoint4[12744] = {X 202.4125, Y 45.3791, Z -5.5000, A 0.000, B 0.000, C 0.000 }
gfCNCPoint4[12745] = {X 201.7358, Y 45.8215, Z -5.5000, A 0.000, B 0.000, C 0.000 }
gfCNCPoint4[12746] = {X 200.9841, Y 46.1192, Z -5.5000, A 0.000, B 0.000, C 0.000 }
gfCNCPoint4[12747] = {X 200.1880, Y 46.2601, Z -5.5000, A 0.000, B 0.000, C 0.000 }
gfCNCPoint4[12748] = {X 199.3798, Y 46.2385, Z -5.5000, A 0.000, B 0.000, C 0.000 }
gfCNCPoint4[12749] = {X 198.5924, Y 46.0553, Z -5.5000, A 0.000, B 0.000, C 0.000 }
gfCNCPoint4[12750] = {X 196.4682, Y 47.1747, Z -5.5000, A 0.000, B 0.000, C 0.000 }
gfCNCPoint4[12751] = {X 194.2562, Y 48.1086, Z -5.5000, A 0.000, B 0.000, C 0.000 }
gfCNCPoint4[12752] = {X 191.9725, Y 48.8502, Z -5.5000, A 0.000, B 0.000, C 0.000 }
gfCNCPoint4[12753] = {X 189.7907, Y 49.3556, Z -5.5000, A 0.000, B 0.000, C 0.000 }
gfCNCPoint4[12754] = {X 187.5689, Y 49.6375, Z -5.5000, A 0.000, B 0.000, C 0.000 }
gfCNCPoint4[12755] = {X 185.3300, Y 49.6929, Z -5.5000, A 0.000, B 0.000, C 0.000 }
gfCNCPoint4[12756] = {X 183.0969, Y 49.5214, Z -5.5000, A 0.000, B 0.000, C 0.000 }
gfCNCPoint4[12757] = {X 180.8928, Y 49.1247, Z -5.5000, A 0.000, B 0.000, C 0.000 }
gfCNCPoint4[12758] = {X 179.0878, Y 48.6016, Z -5.5000, A 0.000, B 0.000, C 0.000 }
gfCNCPoint4[12759] = {X 177.3553, Y 47.8739, Z -5.5000, A 0.000, B 0.000, C 0.000 }
gfCNCPoint4[12760] = {X 175.7181, Y 46.9513, Z -5.5000, A 0.000, B 0.000, C 0.000 }
gfCNCPoint4[12761] = {X 174.1983, Y 45.8461, Z -5.5000, A 0.000, B 0.000, C 0.000 }
gfCNCPoint4[12762] = {X 173.0857, Y 44.8312, Z -5.5000, A 0.000, B 0.000, C 0.000 }
gfCNCPoint4[12763] = {X 172.1010, Y 43.6918, Z -5.5000, A 0.000, B 0.000, C 0.000 }
gfCNCPoint4[12764] = {X 171.2580, Y 42.4439, Z -5.5000, A 0.000, B 0.000, C 0.000 }
gfCNCPoint4[12765] = {X 170.5686, Y 41.1050, Z -5.5000, A 0.000, B 0.000, C 0.000 }
gfCNCPoint4[12766] = {X 170.0425, Y 39.6940, Z -5.5000, A 0.000, B 0.000, C 0.000 }
gfCNCPoint4[12767] = {X 169.6870, Y 38.2306, Z -5.5000, A 0.000, B 0.000, C 0.000 }
gfCNCPoint4[12768] = {X 169.6320, Y 37.8853, Z -5.5000, A 0.000, B 0.000, C 0.000 }
gfCNCPoint4[12769] = {X 165.6027, Y 38.5268, Z -5.5000, A 0.000, B 0.000, C 0.000 }
gfCNCPoint4[12770] = {X 165.6027, Y 38.5268, Z -2.5000, A 0.000, B 0.000, C 0.000 }
gfCNCPoint4[12771] = {X 165.6027, Y 38.5268, Z 11.0000, A 0.000, B 0.000, C 0.000 }
gfCNCPoint4[12772] = {X 210.1645, Y 28.5739, Z 11.0000, A 0.000, B 0.000, C 0.000 }
gfCNCPoint4[12773] = {X 210.1645, Y 28.5739, Z -2.5000, A 0.000, B 0.000, C 0.000 }
gfCNCPoint4[12774] = {X 210.1645, Y 28.5739, Z -5.5000, A 0.000, B 0.000, C 0.000 }
gfCNCPoint4[12775] = {X 214.2445, Y 28.5739, Z -5.5000, A 0.000, B 0.000, C 0.000 }
gfCNCPoint4[12776] = {X 214.2445, Y 17.4625, Z -5.5000, A 0.000, B 0.000, C 0.000 }
gfCNCPoint4[12777] = {X 214.2392, Y 16.7692, Z -5.5000, A 0.000, B 0.000, C 0.000 }
gfCNCPoint4[12778] = {X 214.2425, Y 16.2724, Z -5.5000, A 0.000, B 0.000, C 0.000 }
gfCNCPoint4[12779] = {X 213.6046, Y 15.6012, Z -5.5000, A 0.000, B 0.000, C 0.000 }
gfCNCPoint4[12780] = {X 213.1245, Y 14.8096, Z -5.5000, A 0.000, B 0.000, C 0.000 }
gfCNCPoint4[12781] = {X 212.8241, Y 13.9338, Z -5.5000, A 0.000, B 0.000, C 0.000 }
gfCNCPoint4[12782] = {X 212.7172, Y 13.0141, Z -5.5000, A 0.000, B 0.000, C 0.000 }
gfCNCPoint4[12783] = {X 212.7170, Y 12.1868, Z -5.5000, A 0.000, B 0.000, C 0.000 }
gfCNCPoint4[12784] = {X 212.8253, Y 11.2255, Z -5.5000, A 0.000, B 0.000, C 0.000 }
gfCNCPoint4[12785] = {X 213.1448, Y 10.3124, Z -5.5000, A 0.000, B 0.000, C 0.000 }
gfCNCPoint4[12786] = {X 213.6595, Y 9.4933, Z -5.5000, A 0.000, B 0.000, C 0.000 }
gfCNCPoint4[12787] = {X 214.3435, Y 8.8093, Z -5.5000, A 0.000, B 0.000, C 0.000 }
gfCNCPoint4[12788] = {X 215.1626, Y 8.2946, Z -5.5000, A 0.000, B 0.000, C 0.000 }
gfCNCPoint4[12789] = {X 216.0757, Y 7.9751, Z -5.5000, A 0.000, B 0.000, C 0.000 }
gfCNCPoint4[12790] = {X 217.0370, Y 7.8668, Z -5.5000, A 0.000, B 0.000, C 0.000 }
gfCNCPoint4[12791] = {X 223.4805, Y 7.8668, Z -5.5000, A 0.000, B 0.000, C 0.000 }
gfCNCPoint4[12792] = {X 224.4418, Y 7.9751, Z -5.5000, A 0.000, B 0.000, C 0.000 }
gfCNCPoint4[12793] = {X 225.3549, Y 8.2946, Z -5.5000, A 0.000, B 0.000, C 0.000 }
gfCNCPoint4[12794] = {X 226.1740, Y 8.8093, Z -5.5000, A 0.000, B 0.000, C 0.000 }
gfCNCPoint4[12795] = {X 226.8580, Y 9.4933, Z -5.5000, A 0.000, B 0.000, C 0.000 }
gfCNCPoint4[12796] = {X 227.3727, Y 10.3124, Z -5.5000, A 0.000, B 0.000, C 0.000 }
gfCNCPoint4[12797] = {X 227.6922, Y 11.2255, Z -5.5000, A 0.000, B 0.000, C 0.000 }
gfCNCPoint4[12798] = {X 227.8005, Y 12.1868, Z -5.5000, A 0.000, B 0.000, C 0.000 }
gfCNCPoint4[12799] = {X 227.8005, Y 12.9782, Z -5.5000, A 0.000, B 0.000, C 0.000 }
gfCNCPoint4[12800] = {X 227.6992, Y 13.9080, Z -5.5000, A 0.000, B 0.000, C 0.000 }
gfCNCPoint4[12801] = {X 227.4002, Y 14.7942, Z -5.5000, A 0.000, B 0.000, C 0.000 }
gfCNCPoint4[12802] = {X 226.9174, Y 15.5953, Z -5.5000, A 0.000, B 0.000, C 0.000 }
gfCNCPoint4[12803] = {X 226.2735, Y 16.2737, Z -5.5000, A 0.000, B 0.000, C 0.000 }
gfCNCPoint4[12804] = {X 226.2745, Y 40.9155, Z -5.5000, A 0.000, B 0.000, C 0.000 }
gfCNCPoint4[12805] = {X 226.9117, Y 41.5856, Z -5.5000, A 0.000, B 0.000, C 0.000 }
gfCNCPoint4[12806] = {X 227.3917, Y 42.3760, Z -5.5000, A 0.000, B 0.000, C 0.000 }
gfCNCPoint4[12807] = {X 227.6925, Y 43.2505, Z -5.5000, A 0.000, B 0.000, C 0.000 }
gfCNCPoint4[12808] = {X 227.8003, Y 44.1689, Z -5.5000, A 0.000, B 0.000, C 0.000 }
gfCNCPoint4[12809] = {X 227.8005, Y 45.0000, Z -5.5000, A 0.000, B 0.000, C 0.000 }
gfCNCPoint4[12810] = {X 227.6922, Y 45.9613, Z -5.5000, A 0.000, B 0.000, C 0.000 }
gfCNCPoint4[12811] = {X 227.3727, Y 46.8744, Z -5.5000, A 0.000, B 0.000, C 0.000 }
gfCNCPoint4[12812] = {X 226.8580, Y 47.6935, Z -5.5000, A 0.000, B 0.000, C 0.000 }
gfCNCPoint4[12813] = {X 226.1740, Y 48.3775, Z -5.5000, A 0.000, B 0.000, C 0.000 }
gfCNCPoint4[12814] = {X 225.3549, Y 48.8922, Z -5.5000, A 0.000, B 0.000, C 0.000 }
gfCNCPoint4[12815] = {X 224.4418, Y 49.2117, Z -5.5000, A 0.000, B 0.000, C 0.000 }
gfCNCPoint4[12816] = {X 223.4805, Y 49.3200, Z -5.5000, A 0.000, B 0.000, C 0.000 }
gfCNCPoint4[12817] = {X 217.0370, Y 49.3200, Z -5.5000, A 0.000, B 0.000, C 0.000 }
gfCNCPoint4[12818] = {X 216.0805, Y 49.2128, Z -5.5000, A 0.000, B 0.000, C 0.000 }
gfCNCPoint4[12819] = {X 215.1715, Y 48.8964, Z -5.5000, A 0.000, B 0.000, C 0.000 }
gfCNCPoint4[12820] = {X 214.3551, Y 48.3867, Z -5.5000, A 0.000, B 0.000, C 0.000 }
gfCNCPoint4[12821] = {X 213.6718, Y 47.7088, Z -5.5000, A 0.000, B 0.000, C 0.000 }
gfCNCPoint4[12822] = {X 213.1556, Y 46.8965, Z -5.5000, A 0.000, B 0.000, C 0.000 }
gfCNCPoint4[12823] = {X 212.8320, Y 45.9901, Z -5.5000, A 0.000, B 0.000, C 0.000 }
gfCNCPoint4[12824] = {X 212.7172, Y 45.0345, Z -5.5000, A 0.000, B 0.000, C 0.000 }
gfCNCPoint4[12825] = {X 212.7170, Y 44.1949, Z -5.5000, A 0.000, B 0.000, C 0.000 }
gfCNCPoint4[12826] = {X 212.7888, Y 43.4170, Z -5.5000, A 0.000, B 0.000, C 0.000 }
gfCNCPoint4[12827] = {X 213.0018, Y 42.6653, Z -5.5000, A 0.000, B 0.000, C 0.000 }
gfCNCPoint4[12828] = {X 213.3489, Y 41.9654, Z -5.5000, A 0.000, B 0.000, C 0.000 }
gfCNCPoint4[12829] = {X 213.8182, Y 41.3408, Z -5.5000, A 0.000, B 0.000, C 0.000 }
gfCNCPoint4[12830] = {X 214.2402, Y 40.8754, Z -5.5000, A 0.000, B 0.000, C 0.000 }
gfCNCPoint4[12831] = {X 214.2445, Y 40.3061, Z -5.5000, A 0.000, B 0.000, C 0.000 }
gfCNCPoint4[12832] = {X 214.2445, Y 28.5739, Z -5.5000, A 0.000, B 0.000, C 0.000 }
gfCNCPoint4[12833] = {X 210.2445, Y 28.5739, Z -5.5000, A 0.000, B 0.000, C 0.000 }
gfCNCPoint4[12834] = {X 214.3245, Y 28.5739, Z -5.5000, A 0.000, B 0.000, C 0.000 }
gfCNCPoint4[12835] = {X 214.3245, Y 17.4621, Z -5.5000, A 0.000, B 0.000, C 0.000 }
gfCNCPoint4[12836] = {X 214.3192, Y 16.7692, Z -5.5000, A 0.000, B 0.000, C 0.000 }
gfCNCPoint4[12837] = {X 214.3227, Y 16.2353, Z -5.5000, A 0.000, B 0.000, C 0.000 }
gfCNCPoint4[12838] = {X 213.6852, Y 15.5748, Z -5.5000, A 0.000, B 0.000, C 0.000 }
gfCNCPoint4[12839] = {X 213.2049, Y 14.7925, Z -5.5000, A 0.000, B 0.000, C 0.000 }
gfCNCPoint4[12840] = {X 212.9042, Y 13.9252, Z -5.5000, A 0.000, B 0.000, C 0.000 }
gfCNCPoint4[12841] = {X 212.7972, Y 13.0135, Z -5.5000, A 0.000, B 0.000, C 0.000 }
gfCNCPoint4[12842] = {X 212.7970, Y 12.1868, Z -5.5000, A 0.000, B 0.000, C 0.000 }
gfCNCPoint4[12843] = {X 212.9033, Y 11.2433, Z -5.5000, A 0.000, B 0.000, C 0.000 }
gfCNCPoint4[12844] = {X 213.2169, Y 10.3472, Z -5.5000, A 0.000, B 0.000, C 0.000 }
gfCNCPoint4[12845] = {X 213.7220, Y 9.5432, Z -5.5000, A 0.000, B 0.000, C 0.000 }
gfCNCPoint4[12846] = {X 214.3934, Y 8.8719, Z -5.5000, A 0.000, B 0.000, C 0.000 }
gfCNCPoint4[12847] = {X 215.1973, Y 8.3667, Z -5.5000, A 0.000, B 0.000, C 0.000 }
gfCNCPoint4[12848] = {X 216.0935, Y 8.0531, Z -5.5000, A 0.000, B 0.000, C 0.000 }
gfCNCPoint4[12849] = {X 217.0370, Y 7.9468, Z -5.5000, A 0.000, B 0.000, C 0.000 }
gfCNCPoint4[12850] = {X 223.4805, Y 7.9468, Z -5.5000, A 0.000, B 0.000, C 0.000 }
gfCNCPoint4[12851] = {X 224.4240, Y 8.0531, Z -5.5000, A 0.000, B 0.000, C 0.000 }
gfCNCPoint4[12852] = {X 225.3201, Y 8.3667, Z -5.5000, A 0.000, B 0.000, C 0.000 }
gfCNCPoint4[12853] = {X 226.1241, Y 8.8718, Z -5.5000, A 0.000, B 0.000, C 0.000 }
gfCNCPoint4[12854] = {X 226.7954, Y 9.5432, Z -5.5000, A 0.000, B 0.000, C 0.000 }
gfCNCPoint4[12855] = {X 227.3006, Y 10.3471, Z -5.5000, A 0.000, B 0.000, C 0.000 }
gfCNCPoint4[12856] = {X 227.6142, Y 11.2433, Z -5.5000, A 0.000, B 0.000, C 0.000 }
gfCNCPoint4[12857] = {X 227.7205, Y 12.1868, Z -5.5000, A 0.000, B 0.000, C 0.000 }
gfCNCPoint4[12858] = {X 227.7205, Y 12.9782, Z -5.5000, A 0.000, B 0.000, C 0.000 }
gfCNCPoint4[12859] = {X 227.6191, Y 13.8998, Z -5.5000, A 0.000, B 0.000, C 0.000 }
gfCNCPoint4[12860] = {X 227.3198, Y 14.7773, Z -5.5000, A 0.000, B 0.000, C 0.000 }
gfCNCPoint4[12861] = {X 226.8369, Y 15.5688, Z -5.5000, A 0.000, B 0.000, C 0.000 }
gfCNCPoint4[12862] = {X 226.1935, Y 16.2364, Z -5.5000, A 0.000, B 0.000, C 0.000 }
gfCNCPoint4[12863] = {X 226.1945, Y 40.9528, Z -5.5000, A 0.000, B 0.000, C 0.000 }
gfCNCPoint4[12864] = {X 226.8313, Y 41.6123, Z -5.5000, A 0.000, B 0.000, C 0.000 }
gfCNCPoint4[12865] = {X 227.3114, Y 42.3933, Z -5.5000, A 0.000, B 0.000, C 0.000 }
gfCNCPoint4[12866] = {X 227.6124, Y 43.2593, Z -5.5000, A 0.000, B 0.000, C 0.000 }
gfCNCPoint4[12867] = {X 227.7203, Y 44.1697, Z -5.5000, A 0.000, B 0.000, C 0.000 }
gfCNCPoint4[12868] = {X 227.7205, Y 45.0000, Z -5.5000, A 0.000, B 0.000, C 0.000 }
gfCNCPoint4[12869] = {X 227.6142, Y 45.9435, Z -5.5000, A 0.000, B 0.000, C 0.000 }
gfCNCPoint4[12870] = {X 227.3006, Y 46.8397, Z -5.5000, A 0.000, B 0.000, C 0.000 }
gfCNCPoint4[12871] = {X 226.7954, Y 47.6436, Z -5.5000, A 0.000, B 0.000, C 0.000 }
gfCNCPoint4[12872] = {X 226.1241, Y 48.3150, Z -5.5000, A 0.000, B 0.000, C 0.000 }
gfCNCPoint4[12873] = {X 225.3201, Y 48.8201, Z -5.5000, A 0.000, B 0.000, C 0.000 }
gfCNCPoint4[12874] = {X 224.4240, Y 49.1337, Z -5.5000, A 0.000, B 0.000, C 0.000 }
gfCNCPoint4[12875] = {X 223.4805, Y 49.2400, Z -5.5000, A 0.000, B 0.000, C 0.000 }
gfCNCPoint4[12876] = {X 217.0370, Y 49.2400, Z -5.5000, A 0.000, B 0.000, C 0.000 }
gfCNCPoint4[12877] = {X 216.0982, Y 49.1348, Z -5.5000, A 0.000, B 0.000, C 0.000 }
gfCNCPoint4[12878] = {X 215.2061, Y 48.8243, Z -5.5000, A 0.000, B 0.000, C 0.000 }
gfCNCPoint4[12879] = {X 214.4048, Y 48.3240, Z -5.5000, A 0.000, B 0.000, C 0.000 }
gfCNCPoint4[12880] = {X 213.7341, Y 47.6587, Z -5.5000, A 0.000, B 0.000, C 0.000 }
gfCNCPoint4[12881] = {X 213.2275, Y 46.8614, Z -5.5000, A 0.000, B 0.000, C 0.000 }
gfCNCPoint4[12882] = {X 212.9099, Y 45.9717, Z -5.5000, A 0.000, B 0.000, C 0.000 }
gfCNCPoint4[12883] = {X 212.7972, Y 45.0338, Z -5.5000, A 0.000, B 0.000, C 0.000 }
gfCNCPoint4[12884] = {X 212.7970, Y 44.1949, Z -5.5000, A 0.000, B 0.000, C 0.000 }
gfCNCPoint4[12885] = {X 212.8675, Y 43.4316, Z -5.5000, A 0.000, B 0.000, C 0.000 }
gfCNCPoint4[12886] = {X 213.0765, Y 42.6941, Z -5.5000, A 0.000, B 0.000, C 0.000 }
gfCNCPoint4[12887] = {X 213.4170, Y 42.0074, Z -5.5000, A 0.000, B 0.000, C 0.000 }
gfCNCPoint4[12888] = {X 213.8774, Y 41.3946, Z -5.5000, A 0.000, B 0.000, C 0.000 }
gfCNCPoint4[12889] = {X 214.3199, Y 40.9065, Z -5.5000, A 0.000, B 0.000, C 0.000 }
gfCNCPoint4[12890] = {X 214.3245, Y 40.3065, Z -5.5000, A 0.000, B 0.000, C 0.000 }
gfCNCPoint4[12891] = {X 214.3245, Y 28.5739, Z -5.5000, A 0.000, B 0.000, C 0.000 }
gfCNCPoint4[12892] = {X 210.3245, Y 28.5739, Z -5.5000, A 0.000, B 0.000, C 0.000 }
gfCNCPoint4[12893] = {X 214.4045, Y 28.5739, Z -5.5000, A 0.000, B 0.000, C 0.000 }
gfCNCPoint4[12894] = {X 214.4045, Y 17.4618, Z -5.5000, A 0.000, B 0.000, C 0.000 }
gfCNCPoint4[12895] = {X 214.3992, Y 16.7691, Z -5.5000, A 0.000, B 0.000, C 0.000 }
gfCNCPoint4[12896] = {X 214.4029, Y 16.1978, Z -5.5000, A 0.000, B 0.000, C 0.000 }
gfCNCPoint4[12897] = {X 213.7658, Y 15.5481, Z -5.5000, A 0.000, B 0.000, C 0.000 }
gfCNCPoint4[12898] = {X 213.2853, Y 14.7753, Z -5.5000, A 0.000, B 0.000, C 0.000 }
gfCNCPoint4[12899] = {X 212.9843, Y 13.9165, Z -5.5000, A 0.000, B 0.000, C 0.000 }
gfCNCPoint4[12900] = {X 212.8772, Y 13.0128, Z -5.5000, A 0.000, B 0.000, C 0.000 }
gfCNCPoint4[12901] = {X 212.8770, Y 12.1868, Z -5.5000, A 0.000, B 0.000, C 0.000 }
gfCNCPoint4[12902] = {X 212.9813, Y 11.2611, Z -5.5000, A 0.000, B 0.000, C 0.000 }
gfCNCPoint4[12903] = {X 213.2890, Y 10.3819, Z -5.5000, A 0.000, B 0.000, C 0.000 }
gfCNCPoint4[12904] = {X 213.7846, Y 9.5931, Z -5.5000, A 0.000, B 0.000, C 0.000 }
gfCNCPoint4[12905] = {X 214.4433, Y 8.9344, Z -5.5000, A 0.000, B 0.000, C 0.000 }
gfCNCPoint4[12906] = {X 215.2321, Y 8.4388, Z -5.5000, A 0.000, B 0.000, C 0.000 }
gfCNCPoint4[12907] = {X 216.1113, Y 8.1311, Z -5.5000, A 0.000, B 0.000, C 0.000 }
gfCNCPoint4[12908] = {X 217.0370, Y 8.0268, Z -5.5000, A 0.000, B 0.000, C 0.000 }
gfCNCPoint4[12909] = {X 223.4805, Y 8.0268, Z -5.5000, A 0.000, B 0.000, C 0.000 }
gfCNCPoint4[12910] = {X 224.4062, Y 8.1311, Z -5.5000, A 0.000, B 0.000, C 0.000 }
gfCNCPoint4[12911] = {X 225.2854, Y 8.4388, Z -5.5000, A 0.000, B 0.000, C 0.000 }
gfCNCPoint4[12912] = {X 226.0742, Y 8.9344, Z -5.5000, A 0.000, B 0.000, C 0.000 }
gfCNCPoint4[12913] = {X 226.7329, Y 9.5931, Z -5.5000, A 0.000, B 0.000, C 0.000 }
gfCNCPoint4[12914] = {X 227.2285, Y 10.3819, Z -5.5000, A 0.000, B 0.000, C 0.000 }
gfCNCPoint4[12915] = {X 227.5362, Y 11.2611, Z -5.5000, A 0.000, B 0.000, C 0.000 }
gfCNCPoint4[12916] = {X 227.6405, Y 12.1868, Z -5.5000, A 0.000, B 0.000, C 0.000 }
gfCNCPoint4[12917] = {X 227.6405, Y 12.9782, Z -5.5000, A 0.000, B 0.000, C 0.000 }
gfCNCPoint4[12918] = {X 227.5390, Y 13.8915, Z -5.5000, A 0.000, B 0.000, C 0.000 }
gfCNCPoint4[12919] = {X 227.2394, Y 14.7602, Z -5.5000, A 0.000, B 0.000, C 0.000 }
gfCNCPoint4[12920] = {X 226.7564, Y 15.5420, Z -5.5000, A 0.000, B 0.000, C 0.000 }
gfCNCPoint4[12921] = {X 226.1135, Y 16.1987, Z -5.5000, A 0.000, B 0.000, C 0.000 }
gfCNCPoint4[12922] = {X 226.1145, Y 40.9905, Z -5.5000, A 0.000, B 0.000, C 0.000 }
gfCNCPoint4[12923] = {X 226.7508, Y 41.6393, Z -5.5000, A 0.000, B 0.000, C 0.000 }
gfCNCPoint4[12924] = {X 227.2311, Y 42.4107, Z -5.5000, A 0.000, B 0.000, C 0.000 }
gfCNCPoint4[12925] = {X 227.5324, Y 43.2681, Z -5.5000, A 0.000, B 0.000, C 0.000 }
gfCNCPoint4[12926] = {X 227.6403, Y 44.1704, Z -5.5000, A 0.000, B 0.000, C 0.000 }
gfCNCPoint4[12927] = {X 227.6405, Y 45.0000, Z -5.5000, A 0.000, B 0.000, C 0.000 }
gfCNCPoint4[12928] = {X 227.5362, Y 45.9257, Z -5.5000, A 0.000, B 0.000, C 0.000 }
gfCNCPoint4[12929] = {X 227.2285, Y 46.8050, Z -5.5000, A 0.000, B 0.000, C 0.000 }
gfCNCPoint4[12930] = {X 226.7329, Y 47.5937, Z -5.5000, A 0.000, B 0.000, C 0.000 }
gfCNCPoint4[12931] = {X 226.0742, Y 48.2524, Z -5.5000, A 0.000, B 0.000, C 0.000 }
gfCNCPoint4[12932] = {X 225.2854, Y 48.7480, Z -5.5000, A 0.000, B 0.000, C 0.000 }
gfCNCPoint4[12933] = {X 224.4062, Y 49.0557, Z -5.5000, A 0.000, B 0.000, C 0.000 }
gfCNCPoint4[12934] = {X 223.4805, Y 49.1600, Z -5.5000, A 0.000, B 0.000, C 0.000 }
gfCNCPoint4[12935] = {X 217.0370, Y 49.1600, Z -5.5000, A 0.000, B 0.000, C 0.000 }
gfCNCPoint4[12936] = {X 216.1160, Y 49.0568, Z -5.5000, A 0.000, B 0.000, C 0.000 }
gfCNCPoint4[12937] = {X 215.2406, Y 48.7521, Z -5.5000, A 0.000, B 0.000, C 0.000 }
gfCNCPoint4[12938] = {X 214.4544, Y 48.2613, Z -5.5000, A 0.000, B 0.000, C 0.000 }
gfCNCPoint4[12939] = {X 213.7965, Y 47.6085, Z -5.5000, A 0.000, B 0.000, C 0.000 }
gfCNCPoint4[12940] = {X 213.2993, Y 46.8263, Z -5.5000, A 0.000, B 0.000, C 0.000 }
gfCNCPoint4[12941] = {X 212.9877, Y 45.9534, Z -5.5000, A 0.000, B 0.000, C 0.000 }
gfCNCPoint4[12942] = {X 212.8771, Y 45.0332, Z -5.5000, A 0.000, B 0.000, C 0.000 }
gfCNCPoint4[12943] = {X 212.8770, Y 44.1949, Z -5.5000, A 0.000, B 0.000, C 0.000 }
gfCNCPoint4[12944] = {X 212.9461, Y 43.4462, Z -5.5000, A 0.000, B 0.000, C 0.000 }
gfCNCPoint4[12945] = {X 213.1511, Y 42.7229, Z -5.5000, A 0.000, B 0.000, C 0.000 }
gfCNCPoint4[12946] = {X 213.4851, Y 42.0494, Z -5.5000, A 0.000, B 0.000, C 0.000 }
gfCNCPoint4[12947] = {X 213.9367, Y 41.4483, Z -5.5000, A 0.000, B 0.000, C 0.000 }
gfCNCPoint4[12948] = {X 214.3997, Y 40.9376, Z -5.5000, A 0.000, B 0.000, C 0.000 }
gfCNCPoint4[12949] = {X 214.4045, Y 40.3068, Z -5.5000, A 0.000, B 0.000, C 0.000 }
gfCNCPoint4[12950] = {X 214.4045, Y 28.5739, Z -5.5000, A 0.000, B 0.000, C 0.000 }
gfCNCPoint4[12951] = {X 210.4045, Y 28.5739, Z -5.5000, A 0.000, B 0.000, C 0.000 }
gfCNCPoint4[12952] = {X 214.4845, Y 28.5739, Z -5.5000, A 0.000, B 0.000, C 0.000 }
gfCNCPoint4[12953] = {X 214.4845, Y 17.4614, Z -5.5000, A 0.000, B 0.000, C 0.000 }
gfCNCPoint4[12954] = {X 214.4792, Y 16.7691, Z -5.5000, A 0.000, B 0.000, C 0.000 }
gfCNCPoint4[12955] = {X 214.4832, Y 16.1599, Z -5.5000, A 0.000, B 0.000, C 0.000 }
gfCNCPoint4[12956] = {X 214.4252, Y 16.1125, Z -5.5000, A 0.000, B 0.000, C 0.000 }
gfCNCPoint4[12957] = {X 214.3681, Y 16.0640, Z -5.5000, A 0.000, B 0.000, C 0.000 }
gfCNCPoint4[12958] = {X 213.7777, Y 15.4322, Z -5.5000, A 0.000, B 0.000, C 0.000 }
gfCNCPoint4[12959] = {X 213.3336, Y 14.6902, Z -5.5000, A 0.000, B 0.000, C 0.000 }
gfCNCPoint4[12960] = {X 213.0560, Y 13.8712, Z -5.5000, A 0.000, B 0.000, C 0.000 }
gfCNCPoint4[12961] = {X 212.9572, Y 13.0121, Z -5.5000, A 0.000, B 0.000, C 0.000 }
gfCNCPoint4[12962] = {X 212.9570, Y 12.1868, Z -5.5000, A 0.000, B 0.000, C 0.000 }
gfCNCPoint4[12963] = {X 213.0593, Y 11.2789, Z -5.5000, A 0.000, B 0.000, C 0.000 }
gfCNCPoint4[12964] = {X 213.3611, Y 10.4166, Z -5.5000, A 0.000, B 0.000, C 0.000 }
gfCNCPoint4[12965] = {X 213.8471, Y 9.6430, Z -5.5000, A 0.000, B 0.000, C 0.000 }
gfCNCPoint4[12966] = {X 214.4932, Y 8.9969, Z -5.5000, A 0.000, B 0.000, C 0.000 }
gfCNCPoint4[12967] = {X 215.2668, Y 8.5109, Z -5.5000, A 0.000, B 0.000, C 0.000 }
gfCNCPoint4[12968] = {X 216.1291, Y 8.2091, Z -5.5000, A 0.000, B 0.000, C 0.000 }
gfCNCPoint4[12969] = {X 217.0370, Y 8.1068, Z -5.5000, A 0.000, B 0.000, C 0.000 }
gfCNCPoint4[12970] = {X 223.4805, Y 8.1068, Z -5.5000, A 0.000, B 0.000, C 0.000 }
gfCNCPoint4[12971] = {X 224.3884, Y 8.2091, Z -5.5000, A 0.000, B 0.000, C 0.000 }
gfCNCPoint4[12972] = {X 225.2507, Y 8.5109, Z -5.5000, A 0.000, B 0.000, C 0.000 }
gfCNCPoint4[12973] = {X 226.0243, Y 8.9969, Z -5.5000, A 0.000, B 0.000, C 0.000 }
gfCNCPoint4[12974] = {X 226.6704, Y 9.6430, Z -5.5000, A 0.000, B 0.000, C 0.000 }
gfCNCPoint4[12975] = {X 227.1564, Y 10.4166, Z -5.5000, A 0.000, B 0.000, C 0.000 }
gfCNCPoint4[12976] = {X 227.4582, Y 11.2789, Z -5.5000, A 0.000, B 0.000, C 0.000 }
gfCNCPoint4[12977] = {X 227.5605, Y 12.1868, Z -5.5000, A 0.000, B 0.000, C 0.000 }
gfCNCPoint4[12978] = {X 227.5605, Y 12.9782, Z -5.5000, A 0.000, B 0.000, C 0.000 }
gfCNCPoint4[12979] = {X 227.4588, Y 13.8831, Z -5.5000, A 0.000, B 0.000, C 0.000 }
gfCNCPoint4[12980] = {X 227.1590, Y 14.7430, Z -5.5000, A 0.000, B 0.000, C 0.000 }
gfCNCPoint4[12981] = {X 226.6758, Y 15.5150, Z -5.5000, A 0.000, B 0.000, C 0.000 }
gfCNCPoint4[12982] = {X 226.0335, Y 16.1605, Z -5.5000, A 0.000, B 0.000, C 0.000 }
gfCNCPoint4[12983] = {X 226.0345, Y 41.0284, Z -5.5000, A 0.000, B 0.000, C 0.000 }
gfCNCPoint4[12984] = {X 226.1411, Y 41.1156, Z -5.5000, A 0.000, B 0.000, C 0.000 }
gfCNCPoint4[12985] = {X 226.7343, Y 41.7473, Z -5.5000, A 0.000, B 0.000, C 0.000 }
gfCNCPoint4[12986] = {X 227.1808, Y 42.4901, Z -5.5000, A 0.000, B 0.000, C 0.000 }
gfCNCPoint4[12987] = {X 227.4603, Y 43.3104, Z -5.5000, A 0.000, B 0.000, C 0.000 }
gfCNCPoint4[12988] = {X 227.5603, Y 44.1712, Z -5.5000, A 0.000, B 0.000, C 0.000 }
gfCNCPoint4[12989] = {X 227.5605, Y 45.0000, Z -5.5000, A 0.000, B 0.000, C 0.000 }
gfCNCPoint4[12990] = {X 227.4582, Y 45.9079, Z -5.5000, A 0.000, B 0.000, C 0.000 }
gfCNCPoint4[12991] = {X 227.1564, Y 46.7702, Z -5.5000, A 0.000, B 0.000, C 0.000 }
gfCNCPoint4[12992] = {X 226.6704, Y 47.5438, Z -5.5000, A 0.000, B 0.000, C 0.000 }
gfCNCPoint4[12993] = {X 226.0243, Y 48.1899, Z -5.5000, A 0.000, B 0.000, C 0.000 }
gfCNCPoint4[12994] = {X 225.2507, Y 48.6760, Z -5.5000, A 0.000, B 0.000, C 0.000 }
gfCNCPoint4[12995] = {X 224.3884, Y 48.9777, Z -5.5000, A 0.000, B 0.000, C 0.000 }
gfCNCPoint4[12996] = {X 223.4805, Y 49.0800, Z -5.5000, A 0.000, B 0.000, C 0.000 }
gfCNCPoint4[12997] = {X 217.0370, Y 49.0800, Z -5.5000, A 0.000, B 0.000, C 0.000 }
gfCNCPoint4[12998] = {X 216.1337, Y 48.9787, Z -5.5000, A 0.000, B 0.000, C 0.000 }
gfCNCPoint4[12999] = {X 215.2752, Y 48.6800, Z -5.5000, A 0.000, B 0.000, C 0.000 }
gfCNCPoint4[13000] = {X 214.5041, Y 48.1986, Z -5.5000, A 0.000, B 0.000, C 0.000 }
gfCNCPoint4[13001] = {X 213.8588, Y 47.5584, Z -5.5000, A 0.000, B 0.000, C 0.000 }
gfCNCPoint4[13002] = {X 213.3712, Y 46.7912, Z -5.5000, A 0.000, B 0.000, C 0.000 }
gfCNCPoint4[13003] = {X 213.0656, Y 45.9351, Z -5.5000, A 0.000, B 0.000, C 0.000 }
gfCNCPoint4[13004] = {X 212.9571, Y 45.0325, Z -5.5000, A 0.000, B 0.000, C 0.000 }
gfCNCPoint4[13005] = {X 212.9570, Y 44.1949, Z -5.5000, A 0.000, B 0.000, C 0.000 }
gfCNCPoint4[13006] = {X 213.0248, Y 43.4609, Z -5.5000, A 0.000, B 0.000, C 0.000 }
gfCNCPoint4[13007] = {X 213.2258, Y 42.7517, Z -5.5000, A 0.000, B 0.000, C 0.000 }
gfCNCPoint4[13008] = {X 213.5532, Y 42.0913, Z -5.5000, A 0.000, B 0.000, C 0.000 }
gfCNCPoint4[13009] = {X 213.9960, Y 41.5020, Z -5.5000, A 0.000, B 0.000, C 0.000 }
gfCNCPoint4[13010] = {X 214.4794, Y 40.9687, Z -5.5000, A 0.000, B 0.000, C 0.000 }
gfCNCPoint4[13011] = {X 214.4845, Y 40.3072, Z -5.5000, A 0.000, B 0.000, C 0.000 }
gfCNCPoint4[13012] = {X 214.4845, Y 28.5739, Z -5.5000, A 0.000, B 0.000, C 0.000 }
gfCNCPoint4[13013] = {X 210.4845, Y 28.5739, Z -5.5000, A 0.000, B 0.000, C 0.000 }
gfCNCPoint4[13014] = {X 214.5645, Y 28.5739, Z -5.5000, A 0.000, B 0.000, C 0.000 }
gfCNCPoint4[13015] = {X 214.5645, Y 17.4611, Z -5.5000, A 0.000, B 0.000, C 0.000 }
gfCNCPoint4[13016] = {X 214.5592, Y 16.7687, Z -5.5000, A 0.000, B 0.000, C 0.000 }
gfCNCPoint4[13017] = {X 214.5586, Y 16.1868, Z -5.5000, A 0.000, B 0.000, C 0.000 }
gfCNCPoint4[13018] = {X 214.5756, Y 16.1310, Z -5.5000, A 0.000, B 0.000, C 0.000 }
gfCNCPoint4[13019] = {X 214.4972, Y 16.0682, Z -5.5000, A 0.000, B 0.000, C 0.000 }
gfCNCPoint4[13020] = {X 214.4204, Y 16.0035, Z -5.5000, A 0.000, B 0.000, C 0.000 }
gfCNCPoint4[13021] = {X 213.8365, Y 15.3774, Z -5.5000, A 0.000, B 0.000, C 0.000 }
gfCNCPoint4[13022] = {X 213.3993, Y 14.6414, Z -5.5000, A 0.000, B 0.000, C 0.000 }
gfCNCPoint4[13023] = {X 213.1286, Y 13.8292, Z -5.5000, A 0.000, B 0.000, C 0.000 }
gfCNCPoint4[13024] = {X 213.0370, Y 12.9780, Z -5.5000, A 0.000, B 0.000, C 0.000 }
gfCNCPoint4[13025] = {X 213.0370, Y 12.1868, Z -5.5000, A 0.000, B 0.000, C 0.000 }
gfCNCPoint4[13026] = {X 213.1373, Y 11.2967, Z -5.5000, A 0.000, B 0.000, C 0.000 }
gfCNCPoint4[13027] = {X 213.4331, Y 10.4513, Z -5.5000, A 0.000, B 0.000, C 0.000 }
gfCNCPoint4[13028] = {X 213.9097, Y 9.6929, Z -5.5000, A 0.000, B 0.000, C 0.000 }
gfCNCPoint4[13029] = {X 214.5431, Y 9.0595, Z -5.5000, A 0.000, B 0.000, C 0.000 }
gfCNCPoint4[13030] = {X 215.3015, Y 8.5829, Z -5.5000, A 0.000, B 0.000, C 0.000 }
gfCNCPoint4[13031] = {X 216.1469, Y 8.2871, Z -5.5000, A 0.000, B 0.000, C 0.000 }
gfCNCPoint4[13032] = {X 217.0370, Y 8.1868, Z -5.5000, A 0.000, B 0.000, C 0.000 }
gfCNCPoint4[13033] = {X 223.4805, Y 8.1868, Z -5.5000, A 0.000, B 0.000, C 0.000 }
gfCNCPoint4[13034] = {X 224.3706, Y 8.2871, Z -5.5000, A 0.000, B 0.000, C 0.000 }
gfCNCPoint4[13035] = {X 225.2160, Y 8.5829, Z -5.5000, A 0.000, B 0.000, C 0.000 }
gfCNCPoint4[13036] = {X 225.9744, Y 9.0595, Z -5.5000, A 0.000, B 0.000, C 0.000 }
gfCNCPoint4[13037] = {X 226.6078, Y 9.6929, Z -5.5000, A 0.000, B 0.000, C 0.000 }
gfCNCPoint4[13038] = {X 227.0844, Y 10.4513, Z -5.5000, A 0.000, B 0.000, C 0.000 }
gfCNCPoint4[13039] = {X 227.3802, Y 11.2967, Z -5.5000, A 0.000, B 0.000, C 0.000 }
gfCNCPoint4[13040] = {X 227.4805, Y 12.1868, Z -5.5000, A 0.000, B 0.000, C 0.000 }
gfCNCPoint4[13041] = {X 227.4803, Y 13.0192, Z -5.5000, A 0.000, B 0.000, C 0.000 }
gfCNCPoint4[13042] = {X 227.3717, Y 13.9047, Z -5.5000, A 0.000, B 0.000, C 0.000 }
gfCNCPoint4[13043] = {X 227.0695, Y 14.7441, Z -5.5000, A 0.000, B 0.000, C 0.000 }
gfCNCPoint4[13044] = {X 226.5888, Y 15.4956, Z -5.5000, A 0.000, B 0.000, C 0.000 }
gfCNCPoint4[13045] = {X 225.9535, Y 16.1219, Z -5.5000, A 0.000, B 0.000, C 0.000 }
gfCNCPoint4[13046] = {X 225.9545, Y 41.0663, Z -5.5000, A 0.000, B 0.000, C 0.000 }
gfCNCPoint4[13047] = {X 226.0932, Y 41.1800, Z -5.5000, A 0.000, B 0.000, C 0.000 }
gfCNCPoint4[13048] = {X 226.6787, Y 41.8064, Z -5.5000, A 0.000, B 0.000, C 0.000 }
gfCNCPoint4[13049] = {X 227.1172, Y 42.5431, Z -5.5000, A 0.000, B 0.000, C 0.000 }
gfCNCPoint4[13050] = {X 227.3886, Y 43.3564, Z -5.5000, A 0.000, B 0.000, C 0.000 }
gfCNCPoint4[13051] = {X 227.4805, Y 44.2089, Z -5.5000, A 0.000, B 0.000, C 0.000 }
gfCNCPoint4[13052] = {X 227.4805, Y 45.0000, Z -5.5000, A 0.000, B 0.000, C 0.000 }
gfCNCPoint4[13053] = {X 227.3802, Y 45.8901, Z -5.5000, A 0.000, B 0.000, C 0.000 }
gfCNCPoint4[13054] = {X 227.0844, Y 46.7355, Z -5.5000, A 0.000, B 0.000, C 0.000 }
gfCNCPoint4[13055] = {X 226.6078, Y 47.4940, Z -5.5000, A 0.000, B 0.000, C 0.000 }
gfCNCPoint4[13056] = {X 225.9744, Y 48.1273, Z -5.5000, A 0.000, B 0.000, C 0.000 }
gfCNCPoint4[13057] = {X 225.2160, Y 48.6039, Z -5.5000, A 0.000, B 0.000, C 0.000 }
gfCNCPoint4[13058] = {X 224.3706, Y 48.8997, Z -5.5000, A 0.000, B 0.000, C 0.000 }
gfCNCPoint4[13059] = {X 223.4805, Y 49.0000, Z -5.5000, A 0.000, B 0.000, C 0.000 }
gfCNCPoint4[13060] = {X 217.0370, Y 49.0000, Z -5.5000, A 0.000, B 0.000, C 0.000 }
gfCNCPoint4[13061] = {X 216.1469, Y 48.8997, Z -5.5000, A 0.000, B 0.000, C 0.000 }
gfCNCPoint4[13062] = {X 215.3015, Y 48.6039, Z -5.5000, A 0.000, B 0.000, C 0.000 }
gfCNCPoint4[13063] = {X 214.5430, Y 48.1273, Z -5.5000, A 0.000, B 0.000, C 0.000 }
gfCNCPoint4[13064] = {X 213.9097, Y 47.4939, Z -5.5000, A 0.000, B 0.000, C 0.000 }
gfCNCPoint4[13065] = {X 213.4331, Y 46.7355, Z -5.5000, A 0.000, B 0.000, C 0.000 }
gfCNCPoint4[13066] = {X 213.1373, Y 45.8901, Z -5.5000, A 0.000, B 0.000, C 0.000 }
gfCNCPoint4[13067] = {X 213.0370, Y 45.0000, Z -5.5000, A 0.000, B 0.000, C 0.000 }
gfCNCPoint4[13068] = {X 213.0370, Y 44.1949, Z -5.5000, A 0.000, B 0.000, C 0.000 }
gfCNCPoint4[13069] = {X 213.1548, Y 43.2400, Z -5.5000, A 0.000, B 0.000, C 0.000 }
gfCNCPoint4[13070] = {X 213.5011, Y 42.3423, Z -5.5000, A 0.000, B 0.000, C 0.000 }
gfCNCPoint4[13071] = {X 214.0552, Y 41.5558, Z -5.5000, A 0.000, B 0.000, C 0.000 }
gfCNCPoint4[13072] = {X 214.5592, Y 40.9999, Z -5.5000, A 0.000, B 0.000, C 0.000 }
gfCNCPoint4[13073] = {X 214.5645, Y 40.3075, Z -5.5000, A 0.000, B 0.000, C 0.000 }
gfCNCPoint4[13074] = {X 214.5645, Y 28.5739, Z -5.5000, A 0.000, B 0.000, C 0.000 }
gfCNCPoint4[13075] = {X 210.4845, Y 28.5739, Z -5.5000, A 0.000, B 0.000, C 0.000 }
gfCNCPoint4[13076] = {X 210.4845, Y 28.5739, Z -2.5000, A 0.000, B 0.000, C 0.000 }
gfCNCPoint4[13077] = {X 210.4845, Y 28.5739, Z 11.0000, A 0.000, B 0.000, C 0.000 }
gfCNCPoint4[13078] = {X 273.6042, Y 28.5936, Z 11.0000, A 0.000, B 0.000, C 0.000 }
gfCNCPoint4[13079] = {X 273.6042, Y 28.5936, Z -2.5000, A 0.000, B 0.000, C 0.000 }
gfCNCPoint4[13080] = {X 273.6042, Y 28.5936, Z -5.5000, A 0.000, B 0.000, C 0.000 }
gfCNCPoint4[13081] = {X 269.5242, Y 28.5936, Z -5.5000, A 0.000, B 0.000, C 0.000 }
gfCNCPoint4[13082] = {X 269.5242, Y 40.9137, Z -5.5000, A 0.000, B 0.000, C 0.000 }
gfCNCPoint4[13083] = {X 269.5377, Y 40.9247, Z -5.5000, A 0.000, B 0.000, C 0.000 }
gfCNCPoint4[13084] = {X 270.1700, Y 41.5942, Z -5.5000, A 0.000, B 0.000, C 0.000 }
gfCNCPoint4[13085] = {X 270.6460, Y 42.3825, Z -5.5000, A 0.000, B 0.000, C 0.000 }
gfCNCPoint4[13086] = {X 270.9442, Y 43.2539, Z -5.5000, A 0.000, B 0.000, C 0.000 }
gfCNCPoint4[13087] = {X 271.0508, Y 44.1686, Z -5.5000, A 0.000, B 0.000, C 0.000 }
gfCNCPoint4[13088] = {X 271.0510, Y 45.0000, Z -5.5000, A 0.000, B 0.000, C 0.000 }
gfCNCPoint4[13089] = {X 270.9427, Y 45.9613, Z -5.5000, A 0.000, B 0.000, C 0.000 }
gfCNCPoint4[13090] = {X 270.6232, Y 46.8744, Z -5.5000, A 0.000, B 0.000, C 0.000 }
gfCNCPoint4[13091] = {X 270.1085, Y 47.6935, Z -5.5000, A 0.000, B 0.000, C 0.000 }
gfCNCPoint4[13092] = {X 269.4245, Y 48.3775, Z -5.5000, A 0.000, B 0.000, C 0.000 }
gfCNCPoint4[13093] = {X 268.6054, Y 48.8922, Z -5.5000, A 0.000, B 0.000, C 0.000 }
gfCNCPoint4[13094] = {X 267.6923, Y 49.2117, Z -5.5000, A 0.000, B 0.000, C 0.000 }
gfCNCPoint4[13095] = {X 266.7310, Y 49.3200, Z -5.5000, A 0.000, B 0.000, C 0.000 }
gfCNCPoint4[13096] = {X 260.2876, Y 49.3200, Z -5.5000, A 0.000, B 0.000, C 0.000 }
gfCNCPoint4[13097] = {X 259.3310, Y 49.2128, Z -5.5000, A 0.000, B 0.000, C 0.000 }
gfCNCPoint4[13098] = {X 258.4219, Y 48.8963, Z -5.5000, A 0.000, B 0.000, C 0.000 }
gfCNCPoint4[13099] = {X 257.6054, Y 48.3865, Z -5.5000, A 0.000, B 0.000, C 0.000 }
gfCNCPoint4[13100] = {X 256.9221, Y 47.7085, Z -5.5000, A 0.000, B 0.000, C 0.000 }
gfCNCPoint4[13101] = {X 256.4059, Y 46.8960, Z -5.5000, A 0.000, B 0.000, C 0.000 }
gfCNCPoint4[13102] = {X 256.0824, Y 45.9894, Z -5.5000, A 0.000, B 0.000, C 0.000 }
gfCNCPoint4[13103] = {X 255.9677, Y 45.0336, Z -5.5000, A 0.000, B 0.000, C 0.000 }
gfCNCPoint4[13104] = {X 255.9680, Y 44.1494, Z -5.5000, A 0.000, B 0.000, C 0.000 }
gfCNCPoint4[13105] = {X 256.0784, Y 43.2364, Z -5.5000, A 0.000, B 0.000, C 0.000 }
gfCNCPoint4[13106] = {X 256.3796, Y 42.3675, Z -5.5000, A 0.000, B 0.000, C 0.000 }
gfCNCPoint4[13107] = {X 256.8579, Y 41.5821, Z -5.5000, A 0.000, B 0.000, C 0.000 }
gfCNCPoint4[13108] = {X 257.4915, Y 40.9157, Z -5.5000, A 0.000, B 0.000, C 0.000 }
gfCNCPoint4[13109] = {X 257.4915, Y 34.4738, Z -5.5000, A 0.000, B 0.000, C 0.000 }
gfCNCPoint4[13110] = {X 254.7680, Y 34.4738, Z -5.5000, A 0.000, B 0.000, C 0.000 }
gfCNCPoint4[13111] = {X 250.4838, Y 42.8189, Z -5.5000, A 0.000, B 0.000, C 0.000 }
gfCNCPoint4[13112] = {X 250.6527, Y 43.4864, Z -5.5000, A 0.000, B 0.000, C 0.000 }
gfCNCPoint4[13113] = {X 250.7134, Y 44.1723, Z -5.5000, A 0.000, B 0.000, C 0.000 }
gfCNCPoint4[13114] = {X 250.7136, Y 45.0000, Z -5.5000, A 0.000, B 0.000, C 0.000 }
gfCNCPoint4[13115] = {X 250.6052, Y 45.9613, Z -5.5000, A 0.000, B 0.000, C 0.000 }
gfCNCPoint4[13116] = {X 250.2857, Y 46.8744, Z -5.5000, A 0.000, B 0.000, C 0.000 }
gfCNCPoint4[13117] = {X 249.7711, Y 47.6935, Z -5.5000, A 0.000, B 0.000, C 0.000 }
gfCNCPoint4[13118] = {X 249.0870, Y 48.3775, Z -5.5000, A 0.000, B 0.000, C 0.000 }
gfCNCPoint4[13119] = {X 248.2679, Y 48.8922, Z -5.5000, A 0.000, B 0.000, C 0.000 }
gfCNCPoint4[13120] = {X 247.3548, Y 49.2117, Z -5.5000, A 0.000, B 0.000, C 0.000 }
gfCNCPoint4[13121] = {X 246.3936, Y 49.3200, Z -5.5000, A 0.000, B 0.000, C 0.000 }
gfCNCPoint4[13122] = {X 239.8075, Y 49.3200, Z -5.5000, A 0.000, B 0.000, C 0.000 }
gfCNCPoint4[13123] = {X 238.8462, Y 49.2117, Z -5.5000, A 0.000, B 0.000, C 0.000 }
gfCNCPoint4[13124] = {X 237.9331, Y 48.8922, Z -5.5000, A 0.000, B 0.000, C 0.000 }
gfCNCPoint4[13125] = {X 237.1141, Y 48.3775, Z -5.5000, A 0.000, B 0.000, C 0.000 }
gfCNCPoint4[13126] = {X 236.4300, Y 47.6935, Z -5.5000, A 0.000, B 0.000, C 0.000 }
gfCNCPoint4[13127] = {X 235.9153, Y 46.8744, Z -5.5000, A 0.000, B 0.000, C 0.000 }
gfCNCPoint4[13128] = {X 235.5958, Y 45.9614, Z -5.5000, A 0.000, B 0.000, C 0.000 }
gfCNCPoint4[13129] = {X 235.4875, Y 45.0001, Z -5.5000, A 0.000, B 0.000, C 0.000 }
gfCNCPoint4[13130] = {X 235.4879, Y 44.1494, Z -5.5000, A 0.000, B 0.000, C 0.000 }
gfCNCPoint4[13131] = {X 235.5856, Y 43.2935, Z -5.5000, A 0.000, B 0.000, C 0.000 }
gfCNCPoint4[13132] = {X 235.8511, Y 42.4740, Z -5.5000, A 0.000, B 0.000, C 0.000 }
gfCNCPoint4[13133] = {X 236.2739, Y 41.7236, Z -5.5000, A 0.000, B 0.000, C 0.000 }
gfCNCPoint4[13134] = {X 236.8373, Y 41.0719, Z -5.5000, A 0.000, B 0.000, C 0.000 }
gfCNCPoint4[13135] = {X 237.5187, Y 40.5449, Z -5.5000, A 0.000, B 0.000, C 0.000 }
gfCNCPoint4[13136] = {X 238.2911, Y 40.1637, Z -5.5000, A 0.000, B 0.000, C 0.000 }
gfCNCPoint4[13137] = {X 242.2801, Y 32.3556, Z -5.5000, A 0.000, B 0.000, C 0.000 }
gfCNCPoint4[13138] = {X 241.1101, Y 31.5692, Z -5.5000, A 0.000, B 0.000, C 0.000 }
gfCNCPoint4[13139] = {X 240.0469, Y 30.6434, Z -5.5000, A 0.000, B 0.000, C 0.000 }
gfCNCPoint4[13140] = {X 239.1070, Y 29.5926, Z -5.5000, A 0.000, B 0.000, C 0.000 }
gfCNCPoint4[13141] = {X 238.3050, Y 28.4331, Z -5.5000, A 0.000, B 0.000, C 0.000 }
gfCNCPoint4[13142] = {X 237.6534, Y 27.1829, Z -5.5000, A 0.000, B 0.000, C 0.000 }
gfCNCPoint4[13143] = {X 237.1623, Y 25.8615, Z -5.5000, A 0.000, B 0.000, C 0.000 }
gfCNCPoint4[13144] = {X 236.7421, Y 24.0500, Z -5.5000, A 0.000, B 0.000, C 0.000 }
gfCNCPoint4[13145] = {X 236.5280, Y 22.2028, Z -5.5000, A 0.000, B 0.000, C 0.000 }
gfCNCPoint4[13146] = {X 236.5226, Y 20.3433, Z -5.5000, A 0.000, B 0.000, C 0.000 }
gfCNCPoint4[13147] = {X 236.7261, Y 18.4949, Z -5.5000, A 0.000, B 0.000, C 0.000 }
gfCNCPoint4[13148] = {X 237.1358, Y 16.6811, Z -5.5000, A 0.000, B 0.000, C 0.000 }
gfCNCPoint4[13149] = {X 237.7062, Y 15.1053, Z -5.5000, A 0.000, B 0.000, C 0.000 }
gfCNCPoint4[13150] = {X 238.4933, Y 13.6258, Z -5.5000, A 0.000, B 0.000, C 0.000 }
gfCNCPoint4[13151] = {X 239.4811, Y 12.2721, Z -5.5000, A 0.000, B 0.000, C 0.000 }
gfCNCPoint4[13152] = {X 240.6501, Y 11.0714, Z -5.5000, A 0.000, B 0.000, C 0.000 }
gfCNCPoint4[13153] = {X 241.9768, Y 10.0475, Z -5.5000, A 0.000, B 0.000, C 0.000 }
gfCNCPoint4[13154] = {X 243.4346, Y 9.2211, Z -5.5000, A 0.000, B 0.000, C 0.000 }
gfCNCPoint4[13155] = {X 244.9945, Y 8.6086, Z -5.5000, A 0.000, B 0.000, C 0.000 }
gfCNCPoint4[13156] = {X 246.6252, Y 8.2223, Z -5.5000, A 0.000, B 0.000, C 0.000 }
gfCNCPoint4[13157] = {X 248.7221, Y 7.9508, Z -5.5000, A 0.000, B 0.000, C 0.000 }
gfCNCPoint4[13158] = {X 250.8350, Y 7.8702, Z -5.5000, A 0.000, B 0.000, C 0.000 }
gfCNCPoint4[13159] = {X 266.7633, Y 7.8702, Z -5.5000, A 0.000, B 0.000, C 0.000 }
gfCNCPoint4[13160] = {X 267.7186, Y 7.9850, Z -5.5000, A 0.000, B 0.000, C 0.000 }
gfCNCPoint4[13161] = {X 268.6248, Y 8.3082, Z -5.5000, A 0.000, B 0.000, C 0.000 }
gfCNCPoint4[13162] = {X 269.4370, Y 8.8239, Z -5.5000, A 0.000, B 0.000, C 0.000 }
gfCNCPoint4[13163] = {X 270.1151, Y 9.5065, Z -5.5000, A 0.000, B 0.000, C 0.000 }
gfCNCPoint4[13164] = {X 270.6254, Y 10.3221, Z -5.5000, A 0.000, B 0.000, C 0.000 }
gfCNCPoint4[13165] = {X 270.9426, Y 11.2304, Z -5.5000, A 0.000, B 0.000, C 0.000 }
gfCNCPoint4[13166] = {X 271.0510, Y 12.1864, Z -5.5000, A 0.000, B 0.000, C 0.000 }
gfCNCPoint4[13167] = {X 271.0508, Y 13.0225, Z -5.5000, A 0.000, B 0.000, C 0.000 }
gfCNCPoint4[13168] = {X 270.9425, Y 13.9403, Z -5.5000, A 0.000, B 0.000, C 0.000 }
gfCNCPoint4[13169] = {X 270.6414, Y 14.8141, Z -5.5000, A 0.000, B 0.000, C 0.000 }
gfCNCPoint4[13170] = {X 270.1614, Y 15.6039, Z -5.5000, A 0.000, B 0.000, C 0.000 }
gfCNCPoint4[13171] = {X 269.5243, Y 16.2734, Z -5.5000, A 0.000, B 0.000, C 0.000 }
gfCNCPoint4[13172] = {X 269.5242, Y 28.5936, Z -5.5000, A 0.000, B 0.000, C 0.000 }
gfCNCPoint4[13173] = {X 273.5242, Y 28.5936, Z -5.5000, A 0.000, B 0.000, C 0.000 }
gfCNCPoint4[13174] = {X 269.4442, Y 28.5936, Z -5.5000, A 0.000, B 0.000, C 0.000 }
gfCNCPoint4[13175] = {X 269.4442, Y 40.9517, Z -5.5000, A 0.000, B 0.000, C 0.000 }
gfCNCPoint4[13176] = {X 269.4864, Y 40.9861, Z -5.5000, A 0.000, B 0.000, C 0.000 }
gfCNCPoint4[13177] = {X 270.1067, Y 41.6432, Z -5.5000, A 0.000, B 0.000, C 0.000 }
gfCNCPoint4[13178] = {X 270.5737, Y 42.4168, Z -5.5000, A 0.000, B 0.000, C 0.000 }
gfCNCPoint4[13179] = {X 270.8662, Y 43.2718, Z -5.5000, A 0.000, B 0.000, C 0.000 }
gfCNCPoint4[13180] = {X 270.9708, Y 44.1693, Z -5.5000, A 0.000, B 0.000, C 0.000 }
gfCNCPoint4[13181] = {X 270.9710, Y 45.0000, Z -5.5000, A 0.000, B 0.000, C 0.000 }
gfCNCPoint4[13182] = {X 270.8647, Y 45.9435, Z -5.5000, A 0.000, B 0.000, C 0.000 }
gfCNCPoint4[13183] = {X 270.5511, Y 46.8397, Z -5.5000, A 0.000, B 0.000, C 0.000 }
gfCNCPoint4[13184] = {X 270.0460, Y 47.6436, Z -5.5000, A 0.000, B 0.000, C 0.000 }
gfCNCPoint4[13185] = {X 269.3746, Y 48.3150, Z -5.5000, A 0.000, B 0.000, C 0.000 }
gfCNCPoint4[13186] = {X 268.5707, Y 48.8201, Z -5.5000, A 0.000, B 0.000, C 0.000 }
gfCNCPoint4[13187] = {X 267.6745, Y 49.1337, Z -5.5000, A 0.000, B 0.000, C 0.000 }
gfCNCPoint4[13188] = {X 266.7310, Y 49.2400, Z -5.5000, A 0.000, B 0.000, C 0.000 }
gfCNCPoint4[13189] = {X 260.2876, Y 49.2400, Z -5.5000, A 0.000, B 0.000, C 0.000 }
gfCNCPoint4[13190] = {X 259.3487, Y 49.1347, Z -5.5000, A 0.000, B 0.000, C 0.000 }
gfCNCPoint4[13191] = {X 258.4564, Y 48.8242, Z -5.5000, A 0.000, B 0.000, C 0.000 }
gfCNCPoint4[13192] = {X 257.6550, Y 48.3238, Z -5.5000, A 0.000, B 0.000, C 0.000 }
gfCNCPoint4[13193] = {X 256.9844, Y 47.6583, Z -5.5000, A 0.000, B 0.000, C 0.000 }
gfCNCPoint4[13194] = {X 256.4777, Y 46.8609, Z -5.5000, A 0.000, B 0.000, C 0.000 }
gfCNCPoint4[13195] = {X 256.1603, Y 45.9711, Z -5.5000, A 0.000, B 0.000, C 0.000 }
gfCNCPoint4[13196] = {X 256.0477, Y 45.0330, Z -5.5000, A 0.000, B 0.000, C 0.000 }
gfCNCPoint4[13197] = {X 256.0480, Y 44.1505, Z -5.5000, A 0.000, B 0.000, C 0.000 }
gfCNCPoint4[13198] = {X 256.1585, Y 43.2454, Z -5.5000, A 0.000, B 0.000, C 0.000 }
gfCNCPoint4[13199] = {X 256.4599, Y 42.3850, Z -5.5000, A 0.000, B 0.000, C 0.000 }
gfCNCPoint4[13200] = {X 256.9383, Y 41.6088, Z -5.5000, A 0.000, B 0.000, C 0.000 }
gfCNCPoint4[13201] = {X 257.5715, Y 40.9529, Z -5.5000, A 0.000, B 0.000, C 0.000 }
gfCNCPoint4[13202] = {X 257.5715, Y 34.3938, Z -5.5000, A 0.000, B 0.000, C 0.000 }
gfCNCPoint4[13203] = {X 254.7192, Y 34.3938, Z -5.5000, A 0.000, B 0.000, C 0.000 }
gfCNCPoint4[13204] = {X 250.3971, Y 42.8126, Z -5.5000, A 0.000, B 0.000, C 0.000 }
gfCNCPoint4[13205] = {X 250.5710, Y 43.4831, Z -5.5000, A 0.000, B 0.000, C 0.000 }
gfCNCPoint4[13206] = {X 250.6334, Y 44.1730, Z -5.5000, A 0.000, B 0.000, C 0.000 }
gfCNCPoint4[13207] = {X 250.6336, Y 45.0000, Z -5.5000, A 0.000, B 0.000, C 0.000 }
gfCNCPoint4[13208] = {X 250.5273, Y 45.9435, Z -5.5000, A 0.000, B 0.000, C 0.000 }
gfCNCPoint4[13209] = {X 250.2137, Y 46.8397, Z -5.5000, A 0.000, B 0.000, C 0.000 }
gfCNCPoint4[13210] = {X 249.7085, Y 47.6436, Z -5.5000, A 0.000, B 0.000, C 0.000 }
gfCNCPoint4[13211] = {X 249.0372, Y 48.3150, Z -5.5000, A 0.000, B 0.000, C 0.000 }
gfCNCPoint4[13212] = {X 248.2332, Y 48.8201, Z -5.5000, A 0.000, B 0.000, C 0.000 }
gfCNCPoint4[13213] = {X 247.3370, Y 49.1337, Z -5.5000, A 0.000, B 0.000, C 0.000 }
gfCNCPoint4[13214] = {X 246.3936, Y 49.2400, Z -5.5000, A 0.000, B 0.000, C 0.000 }
gfCNCPoint4[13215] = {X 239.8075, Y 49.2400, Z -5.5000, A 0.000, B 0.000, C 0.000 }
gfCNCPoint4[13216] = {X 238.8640, Y 49.1337, Z -5.5000, A 0.000, B 0.000, C 0.000 }
gfCNCPoint4[13217] = {X 237.9679, Y 48.8201, Z -5.5000, A 0.000, B 0.000, C 0.000 }
gfCNCPoint4[13218] = {X 237.1639, Y 48.3150, Z -5.5000, A 0.000, B 0.000, C 0.000 }
gfCNCPoint4[13219] = {X 236.4926, Y 47.6436, Z -5.5000, A 0.000, B 0.000, C 0.000 }
gfCNCPoint4[13220] = {X 235.9874, Y 46.8397, Z -5.5000, A 0.000, B 0.000, C 0.000 }
gfCNCPoint4[13221] = {X 235.6738, Y 45.9436, Z -5.5000, A 0.000, B 0.000, C 0.000 }
gfCNCPoint4[13222] = {X 235.5675, Y 45.0001, Z -5.5000, A 0.000, B 0.000, C 0.000 }
gfCNCPoint4[13223] = {X 235.5679, Y 44.1505, Z -5.5000, A 0.000, B 0.000, C 0.000 }
gfCNCPoint4[13224] = {X 235.6649, Y 43.3054, Z -5.5000, A 0.000, B 0.000, C 0.000 }
gfCNCPoint4[13225] = {X 235.9285, Y 42.4967, Z -5.5000, A 0.000, B 0.000, C 0.000 }
gfCNCPoint4[13226] = {X 236.3483, Y 41.7570, Z -5.5000, A 0.000, B 0.000, C 0.000 }
gfCNCPoint4[13227] = {X 236.9073, Y 41.1158, Z -5.5000, A 0.000, B 0.000, C 0.000 }
gfCNCPoint4[13228] = {X 237.5830, Y 40.5992, Z -5.5000, A 0.000, B 0.000, C 0.000 }
gfCNCPoint4[13229] = {X 238.3482, Y 40.2278, Z -5.5000, A 0.000, B 0.000, C 0.000 }
gfCNCPoint4[13230] = {X 242.3859, Y 32.3245, Z -5.5000, A 0.000, B 0.000, C 0.000 }
gfCNCPoint4[13231] = {X 241.2088, Y 31.5439, Z -5.5000, A 0.000, B 0.000, C 0.000 }
gfCNCPoint4[13232] = {X 240.1390, Y 30.6217, Z -5.5000, A 0.000, B 0.000, C 0.000 }
gfCNCPoint4[13233] = {X 239.1933, Y 29.5727, Z -5.5000, A 0.000, B 0.000, C 0.000 }
gfCNCPoint4[13234] = {X 238.3866, Y 28.4133, Z -5.5000, A 0.000, B 0.000, C 0.000 }
gfCNCPoint4[13235] = {X 237.7316, Y 27.1620, Z -5.5000, A 0.000, B 0.000, C 0.000 }
gfCNCPoint4[13236] = {X 237.2388, Y 25.8383, Z -5.5000, A 0.000, B 0.000, C 0.000 }
gfCNCPoint4[13237] = {X 236.8208, Y 24.0357, Z -5.5000, A 0.000, B 0.000, C 0.000 }
gfCNCPoint4[13238] = {X 236.6078, Y 22.1976, Z -5.5000, A 0.000, B 0.000, C 0.000 }
gfCNCPoint4[13239] = {X 236.6025, Y 20.3472, Z -5.5000, A 0.000, B 0.000, C 0.000 }
gfCNCPoint4[13240] = {X 236.8050, Y 18.5079, Z -5.5000, A 0.000, B 0.000, C 0.000 }
gfCNCPoint4[13241] = {X 237.2127, Y 16.7030, Z -5.5000, A 0.000, B 0.000, C 0.000 }
gfCNCPoint4[13242] = {X 237.7793, Y 15.1378, Z -5.5000, A 0.000, B 0.000, C 0.000 }
gfCNCPoint4[13243] = {X 238.5611, Y 13.6682, Z -5.5000, A 0.000, B 0.000, C 0.000 }
gfCNCPoint4[13244] = {X 239.5423, Y 12.3236, Z -5.5000, A 0.000, B 0.000, C 0.000 }
gfCNCPoint4[13245] = {X 240.7035, Y 11.1309, Z -5.5000, A 0.000, B 0.000, C 0.000 }
gfCNCPoint4[13246] = {X 242.0213, Y 10.1140, Z -5.5000, A 0.000, B 0.000, C 0.000 }
gfCNCPoint4[13247] = {X 243.4694, Y 9.2931, Z -5.5000, A 0.000, B 0.000, C 0.000 }
gfCNCPoint4[13248] = {X 245.0188, Y 8.6848, Z -5.5000, A 0.000, B 0.000, C 0.000 }
gfCNCPoint4[13249] = {X 246.6386, Y 8.3011, Z -5.5000, A 0.000, B 0.000, C 0.000 }
gfCNCPoint4[13250] = {X 248.7286, Y 8.0305, Z -5.5000, A 0.000, B 0.000, C 0.000 }
gfCNCPoint4[13251] = {X 250.8346, Y 7.9502, Z -5.5000, A 0.000, B 0.000, C 0.000 }
gfCNCPoint4[13252] = {X 266.7627, Y 7.9502, Z -5.5000, A 0.000, B 0.000, C 0.000 }
gfCNCPoint4[13253] = {X 267.7003, Y 8.0629, Z -5.5000, A 0.000, B 0.000, C 0.000 }
gfCNCPoint4[13254] = {X 268.5897, Y 8.3801, Z -5.5000, A 0.000, B 0.000, C 0.000 }
gfCNCPoint4[13255] = {X 269.3869, Y 8.8863, Z -5.5000, A 0.000, B 0.000, C 0.000 }
gfCNCPoint4[13256] = {X 270.0524, Y 9.5562, Z -5.5000, A 0.000, B 0.000, C 0.000 }
gfCNCPoint4[13257] = {X 270.5532, Y 10.3567, Z -5.5000, A 0.000, B 0.000, C 0.000 }
gfCNCPoint4[13258] = {X 270.8646, Y 11.2482, Z -5.5000, A 0.000, B 0.000, C 0.000 }
gfCNCPoint4[13259] = {X 270.9710, Y 12.1865, Z -5.5000, A 0.000, B 0.000, C 0.000 }
gfCNCPoint4[13260] = {X 270.9708, Y 13.0217, Z -5.5000, A 0.000, B 0.000, C 0.000 }
gfCNCPoint4[13261] = {X 270.8624, Y 13.9315, Z -5.5000, A 0.000, B 0.000, C 0.000 }
gfCNCPoint4[13262] = {X 270.5611, Y 14.7968, Z -5.5000, A 0.000, B 0.000, C 0.000 }
gfCNCPoint4[13263] = {X 270.0810, Y 15.5772, Z -5.5000, A 0.000, B 0.000, C 0.000 }
gfCNCPoint4[13264] = {X 269.4443, Y 16.2362, Z -5.5000, A 0.000, B 0.000, C 0.000 }
gfCNCPoint4[13265] = {X 269.4442, Y 28.5936, Z -5.5000, A 0.000, B 0.000, C 0.000 }
gfCNCPoint4[13266] = {X 273.4442, Y 28.5936, Z -5.5000, A 0.000, B 0.000, C 0.000 }
gfCNCPoint4[13267] = {X 269.3642, Y 28.5936, Z -5.5000, A 0.000, B 0.000, C 0.000 }
gfCNCPoint4[13268] = {X 269.3642, Y 40.9897, Z -5.5000, A 0.000, B 0.000, C 0.000 }
gfCNCPoint4[13269] = {X 269.4351, Y 41.0475, Z -5.5000, A 0.000, B 0.000, C 0.000 }
gfCNCPoint4[13270] = {X 270.0434, Y 41.6921, Z -5.5000, A 0.000, B 0.000, C 0.000 }
gfCNCPoint4[13271] = {X 270.5014, Y 42.4510, Z -5.5000, A 0.000, B 0.000, C 0.000 }
gfCNCPoint4[13272] = {X 270.7882, Y 43.2897, Z -5.5000, A 0.000, B 0.000, C 0.000 }
